SPLINE
SPL {X  -123.821, Y  +785.537, Z    +0.000, E1   -64.536, E3 +26761.912}
SPL {X  -153.467, Y  +737.853, Z    +0.000, E1   -51.757, E3 +26764.227}
SPL {X  -161.000, Y  +714.475, Z    +0.000, E1   -39.424, E3 +26763.699}
SPL {X  -164.534, Y  +694.695, Z    +0.000, E1   -23.511, E3 +26761.989}
SPL {X  -165.597, Y  +679.703, Z    +0.000, E1    -7.645, E3 +26761.865}
SPL {X  -165.650, Y  +673.520, Z    +0.000, E1    -0.048, E3 +26760.817}
SPL {X  -165.650, Y  +671.692, Z    +0.000, E1    +4.450, E3 +26760.383}
SPL {X  -165.650, Y  +667.743, Z    +0.000, E1   +15.617, E3 +26760.301}
SPL {X  -165.650, Y  +662.891, Z    +0.000, E1   +29.740, E3 +26759.819}
SPL {X  -165.650, Y  +658.373, Z    +0.000, E1   +40.877, E3 +26760.016}
SPL {X  -165.650, Y  +650.834, Z    +0.000, E1   +55.143, E3 +26759.270}
SPL {X  -165.650, Y  +639.785, Z    +0.000, E1   +67.512, E3 +26758.487}
SPL {X  -165.650, Y  +619.979, Z    +0.000, E1   +79.465, E3 +26754.656}
SPL {X  -165.650, Y  +584.722, Z    +0.000, E1   +79.551, E3 +26763.947}
SPL {X  -165.650, Y  +560.326, Z    +0.000, E1   +78.360, E3 +26773.669}
SPL {X  -160.258, Y  +336.579, Z    +0.000, E1   +78.314, E3 +26845.191}
SPL {X  -159.618, Y  +334.207, Z    +0.000, E1   +75.622, E3 +26876.005}
SPL {X  -156.487, Y  +324.170, Z    +0.000, E1   +75.150, E3 +26886.360}
SPL {X  -142.256, Y  +293.629, Z    +0.000, E1   +77.020, E3 +26881.460}
ENDSPLINE

SPLINE
SPL {X  -142.811, Y  +294.566, Z    +0.000, E1   +75.668, E3 +26893.422}
ENDSPLINE

SPLINE
SPL {X  -141.646, Y  +292.615, Z    +0.000, E1   +74.702, E3 +26902.516}
SPL {X  -140.419, Y  +290.622, Z    +0.000, E1   +73.705, E3 +26911.359}
SPL {X  -136.008, Y  +283.940, Z    +0.000, E1   +73.594, E3 +26915.478}
SPL {X  -132.748, Y  +279.415, Z    +0.000, E1   +73.006, E3 +26921.534}
SPL {X  -129.007, Y  +274.590, Z    +0.000, E1   +72.484, E3 +26926.883}
SPL {X  -125.914, Y  +270.864, Z    +0.000, E1   +72.144, E3 +26930.375}
SPL {X  -123.729, Y  +268.359, Z    +0.000, E1   +71.932, E3 +26932.547}
SPL {X  -111.023, Y  +255.562, Z    +0.000, E1   +75.772, E3 +26923.413}
SPL {X   -49.289, Y  +220.353, Z    +0.000, E1   +56.690, E3 +27116.128}
ENDSPLINE

SPLINE
SPL {X  -127.117, Y  +272.287, Z    +0.000, E1   +62.713, E3 +27285.350}
SPL {X  -154.956, Y  +319.945, Z    +0.000, E1   +49.402, E3 +27289.749}
SPL {X  -162.871, Y  +348.286, Z    +0.000, E1   +32.462, E3 +27288.776}
SPL {X  -165.127, Y  +365.342, Z    +0.000, E1   +17.250, E3 +27288.615}
SPL {X  -165.640, Y  +376.693, Z    +0.000, E1    +4.721, E3 +27288.188}
SPL {X  -165.650, Y  +380.500, Z    +0.000, E1    -0.000, E3 +27287.339}
SPL {X  -165.650, Y  +382.123, Z    +0.000, E1    -3.912, E3 +27286.966}
SPL {X  -165.650, Y  +387.069, Z    +0.000, E1   -17.420, E3 +27286.677}
SPL {X  -165.650, Y  +393.439, Z    +0.000, E1   -35.398, E3 +27286.223}
SPL {X  -165.650, Y  +400.610, Z    +0.000, E1   -50.510, E3 +27285.961}
SPL {X  -165.650, Y  +414.376, Z    +0.000, E1   -68.098, E3 +27283.994}
SPL {X  -165.650, Y  +468.582, Z    +0.000, E1   -78.237, E3 +27292.765}
SPL {X  -160.244, Y  +717.475, Z    +0.000, E1   -78.917, E3 +27365.322}
SPL {X  -159.651, Y  +719.676, Z    +0.000, E1   -75.661, E3 +27401.709}
SPL {X  -157.156, Y  +727.862, Z    +0.000, E1   -75.175, E3 +27411.191}
SPL {X  -154.068, Y  +736.353, Z    +0.000, E1   -74.906, E3 +27418.366}
SPL {X  -149.738, Y  +746.340, Z    +0.000, E1   -74.451, E3 +27428.054}
SPL {X  -144.163, Y  +757.090, Z    +0.000, E1   -74.033, E3 +27437.146}
SPL {X  -139.284, Y  +765.165, Z    +0.000, E1   -73.322, E3 +27446.841}
SPL {X  -134.662, Y  +771.969, Z    +0.000, E1   -72.884, E3 +27453.173}
SPL {X  -131.459, Y  +776.289, Z    +0.000, E1   -72.475, E3 +27457.840}
SPL {X  -127.605, Y  +781.126, Z    +0.000, E1   -71.922, E3 +27463.284}
SPL {X  -124.773, Y  +784.457, Z    +0.000, E1   -71.383, E3 +27467.331}
SPL {X  -119.086, Y  +790.645, Z    +0.000, E1   -72.931, E3 +27464.185}
SPL {X   -51.449, Y  +832.958, Z    +0.000, E1   -57.230, E3 +27621.705}
ENDSPLINE

SPLINE
SPL {X  -123.821, Y  +785.537, Z    +0.000, E1   -64.536, E3 +27823.450}
SPL {X  -153.467, Y  +737.853, Z    +0.000, E1   -51.757, E3 +27825.765}
SPL {X  -161.000, Y  +714.475, Z    +0.000, E1   -39.424, E3 +27825.238}
SPL {X  -164.534, Y  +694.695, Z    +0.000, E1   -23.511, E3 +27823.528}
SPL {X  -165.597, Y  +679.703, Z    +0.000, E1    -7.645, E3 +27823.403}
SPL {X  -165.650, Y  +673.520, Z    +0.000, E1    -0.048, E3 +27822.355}
SPL {X  -165.650, Y  +671.692, Z    +0.000, E1    +4.450, E3 +27821.922}
SPL {X  -165.650, Y  +667.743, Z    +0.000, E1   +15.617, E3 +27821.840}
SPL {X  -165.650, Y  +661.459, Z    +0.000, E1   +33.218, E3 +27821.420}
SPL {X  -165.650, Y  +653.296, Z    +0.000, E1   +51.333, E3 +27820.975}
SPL {X  -165.650, Y  +642.000, Z    +0.000, E1   +65.561, E3 +27820.188}
SPL {X  -165.650, Y  +619.979, Z    +0.000, E1   +79.465, E3 +27816.194}
SPL {X  -165.650, Y  +569.632, Z    +0.000, E1   +78.783, E3 +27831.473}
SPL {X  -158.840, Y  +331.491, Z    +0.000, E1   +77.462, E3 +27917.783}
ENDSPLINE

SPLINE
SPL {X  -159.893, Y  +335.208, Z    +0.000, E1   +75.483, E3 +27938.518}
ENDSPLINE

SPLINE
SPL {X  -156.487, Y  +324.170, Z    +0.000, E1   +75.150, E3 +27947.899}
SPL {X  -142.256, Y  +293.629, Z    +0.000, E1   +77.020, E3 +27942.999}
ENDSPLINE

SPLINE
SPL {X  -142.811, Y  +294.566, Z    +0.000, E1   +75.668, E3 +27954.961}
ENDSPLINE

SPLINE
SPL {X  -141.646, Y  +292.615, Z    +0.000, E1   +74.702, E3 +27964.055}
SPL {X  -140.419, Y  +290.622, Z    +0.000, E1   +73.705, E3 +27972.898}
SPL {X  -136.008, Y  +283.940, Z    +0.000, E1   +73.594, E3 +27977.017}
SPL {X  -132.748, Y  +279.415, Z    +0.000, E1   +73.006, E3 +27983.073}
SPL {X  -129.007, Y  +274.590, Z    +0.000, E1   +72.484, E3 +27988.421}
SPL {X  -125.914, Y  +270.864, Z    +0.000, E1   +72.144, E3 +27991.913}
SPL {X  -123.729, Y  +268.359, Z    +0.000, E1   +71.932, E3 +27994.085}
SPL {X  -111.023, Y  +255.562, Z    +0.000, E1   +75.772, E3 +27984.951}
SPL {X   -49.289, Y  +220.353, Z    +0.000, E1   +56.690, E3 +28177.666}
ENDSPLINE

SPLINE
SPL {X  -127.117, Y  +272.287, Z    +0.000, E1   +62.713, E3 +28346.888}
SPL {X  -154.956, Y  +319.945, Z    +0.000, E1   +49.402, E3 +28351.287}
SPL {X  -162.871, Y  +348.286, Z    +0.000, E1   +32.462, E3 +28350.315}
SPL {X  -165.127, Y  +365.342, Z    +0.000, E1   +17.250, E3 +28350.153}
SPL {X  -165.640, Y  +376.693, Z    +0.000, E1    +4.721, E3 +28349.726}
SPL {X  -165.650, Y  +380.500, Z    +0.000, E1    -0.000, E3 +28348.877}
SPL {X  -165.650, Y  +383.262, Z    +0.000, E1    -6.645, E3 +28348.406}
SPL {X  -165.650, Y  +388.390, Z    +0.000, E1   -21.508, E3 +28348.194}
SPL {X  -165.650, Y  +393.439, Z    +0.000, E1   -35.398, E3 +28347.762}
SPL {X  -165.650, Y  +400.610, Z    +0.000, E1   -50.510, E3 +28347.499}
SPL {X  -165.650, Y  +414.376, Z    +0.000, E1   -68.098, E3 +28345.533}
SPL {X  -165.650, Y  +468.582, Z    +0.000, E1   -78.237, E3 +28354.303}
SPL {X  -158.306, Y  +724.277, Z    +0.000, E1   -77.461, E3 +28444.744}
ENDSPLINE

SPLINE
SPL {X  -160.145, Y  +717.851, Z    +0.000, E1   -75.386, E3 +28465.258}
ENDSPLINE

SPLINE
SPL {X  -157.156, Y  +727.862, Z    +0.000, E1   -75.175, E3 +28472.730}
SPL {X  -154.068, Y  +736.353, Z    +0.000, E1   -74.906, E3 +28479.905}
SPL {X  -149.738, Y  +746.340, Z    +0.000, E1   -74.451, E3 +28489.592}
SPL {X  -144.163, Y  +757.090, Z    +0.000, E1   -74.033, E3 +28498.685}
SPL {X  -140.473, Y  +763.291, Z    +0.000, E1   -73.478, E3 +28506.126}
SPL {X  -135.914, Y  +770.196, Z    +0.000, E1   -72.974, E3 +28513.302}
SPL {X  -131.459, Y  +776.289, Z    +0.000, E1   -72.475, E3 +28519.378}
SPL {X  -128.771, Y  +779.702, Z    +0.000, E1   -71.875, E3 +28524.325}
SPL {X  -124.506, Y  +784.762, Z    +0.000, E1   -71.815, E3 +28527.213}
SPL {X  -112.958, Y  +796.663, Z    +0.000, E1   -74.119, E3 +28523.917}
SPL {X   -51.449, Y  +832.958, Z    +0.000, E1   -57.230, E3 +28683.244}
ENDSPLINE

SPLINE
SPL {X  -123.821, Y  +785.537, Z    +0.000, E1   -64.536, E3 +28884.989}
SPL {X  -153.467, Y  +737.853, Z    +0.000, E1   -51.757, E3 +28887.304}
SPL {X  -162.176, Y  +709.248, Z    +0.000, E1   -35.773, E3 +28886.329}
SPL {X  -164.888, Y  +691.368, Z    +0.000, E1   -20.174, E3 +28884.767}
SPL {X  -165.597, Y  +679.703, Z    +0.000, E1    -7.645, E3 +28884.942}
SPL {X  -165.650, Y  +673.520, Z    +0.000, E1    -0.048, E3 +28883.894}
SPL {X  -165.650, Y  +671.692, Z    +0.000, E1    +4.450, E3 +28883.460}
SPL {X  -165.650, Y  +667.743, Z    +0.000, E1   +15.617, E3 +28883.378}
SPL {X  -165.650, Y  +661.459, Z    +0.000, E1   +33.218, E3 +28882.959}
SPL {X  -165.650, Y  +650.834, Z    +0.000, E1   +55.143, E3 +28882.347}
SPL {X  -165.650, Y  +639.785, Z    +0.000, E1   +67.512, E3 +28881.564}
SPL {X  -165.650, Y  +619.979, Z    +0.000, E1   +79.465, E3 +28877.733}
SPL {X  -165.650, Y  +569.632, Z    +0.000, E1   +78.783, E3 +28893.011}
SPL {X  -158.840, Y  +331.491, Z    +0.000, E1   +77.462, E3 +28979.322}
ENDSPLINE

SPLINE
SPL {X  -159.893, Y  +335.208, Z    +0.000, E1   +75.483, E3 +29000.056}
ENDSPLINE

SPLINE
SPL {X  -156.487, Y  +324.170, Z    +0.000, E1   +75.150, E3 +29009.437}
SPL {X  -142.256, Y  +293.629, Z    +0.000, E1   +77.020, E3 +29004.537}
ENDSPLINE

SPLINE
SPL {X  -142.811, Y  +294.566, Z    +0.000, E1   +75.668, E3 +29016.499}
ENDSPLINE

SPLINE
SPL {X  -141.646, Y  +292.615, Z    +0.000, E1   +74.702, E3 +29025.593}
SPL {X  -140.419, Y  +290.622, Z    +0.000, E1   +73.705, E3 +29034.436}
SPL {X  -136.008, Y  +283.940, Z    +0.000, E1   +73.594, E3 +29038.555}
SPL {X  -132.748, Y  +279.415, Z    +0.000, E1   +73.006, E3 +29044.611}
SPL {X  -129.007, Y  +274.590, Z    +0.000, E1   +72.484, E3 +29049.960}
SPL {X  -125.914, Y  +270.864, Z    +0.000, E1   +72.144, E3 +29053.451}
SPL {X  -123.729, Y  +268.359, Z    +0.000, E1   +71.932, E3 +29055.624}
SPL {X  -111.023, Y  +255.562, Z    +0.000, E1   +75.772, E3 +29046.490}
SPL {X   -49.289, Y  +220.353, Z    +0.000, E1   +56.690, E3 +29239.205}
ENDSPLINE

SPLINE
SPL {X  -127.117, Y  +272.287, Z    +0.000, E1   +62.713, E3 +29408.427}
SPL {X  -152.442, Y  +313.682, Z    +0.000, E1   +51.943, E3 +29412.658}
SPL {X  -162.319, Y  +345.447, Z    +0.000, E1   +34.671, E3 +29412.084}
SPL {X  -165.127, Y  +365.342, Z    +0.000, E1   +17.250, E3 +29411.692}
SPL {X  -165.640, Y  +376.693, Z    +0.000, E1    +4.721, E3 +29411.265}
SPL {X  -165.650, Y  +380.500, Z    +0.000, E1    -0.000, E3 +29410.416}
SPL {X  -165.650, Y  +383.262, Z    +0.000, E1    -6.645, E3 +29409.945}
SPL {X  -165.650, Y  +388.390, Z    +0.000, E1   -21.508, E3 +29409.733}
SPL {X  -165.650, Y  +393.439, Z    +0.000, E1   -35.398, E3 +29409.300}
SPL {X  -165.650, Y  +400.610, Z    +0.000, E1   -50.510, E3 +29409.038}
SPL {X  -165.650, Y  +414.376, Z    +0.000, E1   -68.098, E3 +29407.071}
SPL {X  -165.650, Y  +459.729, Z    +0.000, E1   -78.035, E3 +29413.526}
SPL {X  -165.650, Y  +475.450, Z    +0.000, E1   -78.345, E3 +29417.640}
SPL {X  -158.306, Y  +724.277, Z    +0.000, E1   -77.461, E3 +29506.283}
ENDSPLINE

SPLINE
SPL {X  -160.145, Y  +717.851, Z    +0.000, E1   -75.386, E3 +29526.796}
ENDSPLINE

SPLINE
SPL {X  -157.156, Y  +727.862, Z    +0.000, E1   -75.175, E3 +29534.268}
SPL {X  -154.068, Y  +736.353, Z    +0.000, E1   -74.906, E3 +29541.443}
SPL {X  -149.738, Y  +746.340, Z    +0.000, E1   -74.451, E3 +29551.131}
SPL {X  -145.204, Y  +755.223, Z    +0.000, E1   -74.188, E3 +29557.857}
SPL {X  -141.453, Y  +761.704, Z    +0.000, E1   -73.638, E3 +29565.779}
SPL {X  -135.914, Y  +770.196, Z    +0.000, E1   -72.974, E3 +29574.841}
SPL {X  -131.459, Y  +776.289, Z    +0.000, E1   -72.475, E3 +29580.917}
SPL {X  -128.771, Y  +779.702, Z    +0.000, E1   -71.875, E3 +29585.863}
SPL {X  -124.506, Y  +784.762, Z    +0.000, E1   -71.815, E3 +29588.752}
SPL {X  -112.958, Y  +796.663, Z    +0.000, E1   -74.119, E3 +29585.455}
SPL {X   -51.449, Y  +832.958, Z    +0.000, E1   -57.230, E3 +29744.782}
ENDSPLINE

SPLINE
SPL {X  -123.821, Y  +785.537, Z    +0.000, E1   -64.536, E3 +29946.527}
SPL {X  -153.467, Y  +737.853, Z    +0.000, E1   -51.757, E3 +29948.842}
SPL {X  -162.176, Y  +709.248, Z    +0.000, E1   -35.773, E3 +29947.868}
SPL {X  -164.888, Y  +691.368, Z    +0.000, E1   -20.174, E3 +29946.305}
SPL {X  -165.597, Y  +679.703, Z    +0.000, E1    -7.645, E3 +29946.480}
SPL {X  -165.650, Y  +673.520, Z    +0.000, E1    -0.048, E3 +29945.432}
SPL {X  -165.650, Y  +671.692, Z    +0.000, E1    +4.450, E3 +29944.999}
SPL {X  -165.650, Y  +667.743, Z    +0.000, E1   +15.617, E3 +29944.917}
SPL {X  -165.650, Y  +661.459, Z    +0.000, E1   +33.218, E3 +29944.497}
SPL {X  -165.650, Y  +653.296, Z    +0.000, E1   +51.333, E3 +29944.052}
SPL {X  -165.650, Y  +642.000, Z    +0.000, E1   +65.561, E3 +29943.265}
SPL {X  -165.650, Y  +619.979, Z    +0.000, E1   +79.465, E3 +29939.271}
SPL {X  -165.650, Y  +569.632, Z    +0.000, E1   +78.783, E3 +29954.550}
SPL {X  -158.840, Y  +331.491, Z    +0.000, E1   +77.462, E3 +30040.860}
ENDSPLINE

SPLINE
SPL {X  -159.893, Y  +335.208, Z    +0.000, E1   +75.483, E3 +30061.595}
ENDSPLINE

SPLINE
SPL {X  -156.487, Y  +324.170, Z    +0.000, E1   +75.150, E3 +30070.976}
SPL {X  -142.256, Y  +293.629, Z    +0.000, E1   +77.020, E3 +30066.076}
ENDSPLINE

SPLINE
SPL {X  -142.811, Y  +294.566, Z    +0.000, E1   +75.668, E3 +30078.038}
ENDSPLINE

SPLINE
SPL {X  -141.646, Y  +292.615, Z    +0.000, E1   +74.702, E3 +30087.131}
SPL {X  -140.419, Y  +290.622, Z    +0.000, E1   +73.705, E3 +30095.975}
SPL {X  -135.839, Y  +283.697, Z    +0.000, E1   +73.388, E3 +30101.713}
SPL {X  -131.336, Y  +277.551, Z    +0.000, E1   +72.879, E3 +30107.965}
SPL {X  -126.848, Y  +271.966, Z    +0.000, E1   +72.322, E3 +30113.693}
SPL {X  -123.729, Y  +268.359, Z    +0.000, E1   +71.932, E3 +30117.162}
SPL {X  -111.023, Y  +255.562, Z    +0.000, E1   +75.772, E3 +30108.028}
SPL {X   -52.752, Y  +221.474, Z    +0.000, E1   +59.157, E3 +30237.280}
SPL {X   -49.901, Y  +220.545, Z    +0.000, E1   +56.696, E3 +30323.672}
ENDSPLINE

SPLINE
SPL {X  -127.117, Y  +272.287, Z    +0.000, E1   +62.713, E3 +30469.965}
SPL {X  -152.442, Y  +313.682, Z    +0.000, E1   +51.943, E3 +30474.197}
SPL {X  -162.319, Y  +345.447, Z    +0.000, E1   +34.671, E3 +30473.622}
SPL {X  -165.127, Y  +365.342, Z    +0.000, E1   +17.250, E3 +30473.230}
SPL {X  -165.640, Y  +376.693, Z    +0.000, E1    +4.721, E3 +30472.803}
SPL {X  -165.650, Y  +380.500, Z    +0.000, E1    -0.000, E3 +30471.954}
SPL {X  -165.650, Y  +382.123, Z    +0.000, E1    -3.912, E3 +30471.581}
SPL {X  -165.650, Y  +387.069, Z    +0.000, E1   -17.420, E3 +30471.293}
SPL {X  -165.650, Y  +393.439, Z    +0.000, E1   -35.398, E3 +30470.839}
SPL {X  -165.650, Y  +400.610, Z    +0.000, E1   -50.510, E3 +30470.576}
SPL {X  -165.650, Y  +414.376, Z    +0.000, E1   -68.098, E3 +30468.610}
SPL {X  -165.650, Y  +468.582, Z    +0.000, E1   -78.237, E3 +30477.380}
SPL {X  -160.244, Y  +717.475, Z    +0.000, E1   -78.917, E3 +30549.938}
SPL {X  -159.651, Y  +719.676, Z    +0.000, E1   -75.661, E3 +30586.324}
SPL {X  -157.156, Y  +727.862, Z    +0.000, E1   -75.175, E3 +30595.807}
SPL {X  -154.068, Y  +736.353, Z    +0.000, E1   -74.906, E3 +30602.981}
SPL {X  -149.738, Y  +746.340, Z    +0.000, E1   -74.451, E3 +30612.669}
SPL {X  -144.163, Y  +757.090, Z    +0.000, E1   -74.033, E3 +30621.762}
SPL {X  -139.284, Y  +765.165, Z    +0.000, E1   -73.322, E3 +30631.456}
SPL {X  -134.662, Y  +771.969, Z    +0.000, E1   -72.884, E3 +30637.788}
SPL {X  -131.459, Y  +776.289, Z    +0.000, E1   -72.475, E3 +30642.455}
SPL {X  -127.605, Y  +781.126, Z    +0.000, E1   -71.922, E3 +30647.899}
SPL {X  -124.773, Y  +784.457, Z    +0.000, E1   -71.383, E3 +30651.947}
SPL {X  -119.086, Y  +790.645, Z    +0.000, E1   -72.931, E3 +30648.801}
SPL {X   -51.449, Y  +832.958, Z    +0.000, E1   -57.230, E3 +30806.321}
ENDSPLINE

SPLINE
SPL {X  -123.821, Y  +785.537, Z    +0.000, E1   -64.536, E3 +31008.066}
SPL {X  -153.467, Y  +737.853, Z    +0.000, E1   -51.757, E3 +31010.381}
SPL {X  -161.000, Y  +714.475, Z    +0.000, E1   -39.424, E3 +31009.853}
SPL {X  -164.534, Y  +694.695, Z    +0.000, E1   -23.511, E3 +31008.143}
SPL {X  -165.597, Y  +679.703, Z    +0.000, E1    -7.645, E3 +31008.019}
SPL {X  -165.650, Y  +673.520, Z    +0.000, E1    -0.048, E3 +31006.971}
SPL {X  -165.650, Y  +671.692, Z    +0.000, E1    +4.450, E3 +31006.537}
SPL {X  -165.650, Y  +667.743, Z    +0.000, E1   +15.617, E3 +31006.455}
SPL {X  -165.650, Y  +661.459, Z    +0.000, E1   +33.218, E3 +31006.035}
SPL {X  -165.650, Y  +653.296, Z    +0.000, E1   +51.333, E3 +31005.591}
SPL {X  -165.650, Y  +642.000, Z    +0.000, E1   +65.561, E3 +31004.803}
SPL {X  -165.650, Y  +619.979, Z    +0.000, E1   +79.465, E3 +31000.810}
SPL {X  -165.650, Y  +569.632, Z    +0.000, E1   +78.783, E3 +31016.088}
SPL {X  -158.840, Y  +331.491, Z    +0.000, E1   +77.462, E3 +31102.398}
ENDSPLINE

SPLINE
SPL {X  -159.893, Y  +335.208, Z    +0.000, E1   +75.483, E3 +31123.133}
ENDSPLINE

SPLINE
SPL {X  -156.487, Y  +324.170, Z    +0.000, E1   +75.150, E3 +31132.514}
SPL {X  -142.256, Y  +293.629, Z    +0.000, E1   +77.020, E3 +31127.614}
ENDSPLINE

SPLINE
SPL {X  -142.811, Y  +294.566, Z    +0.000, E1   +75.668, E3 +31139.576}
ENDSPLINE

SPLINE
SPL {X  -141.646, Y  +292.615, Z    +0.000, E1   +74.702, E3 +31148.670}
SPL {X  -140.419, Y  +290.622, Z    +0.000, E1   +73.705, E3 +31157.513}
SPL {X  -136.008, Y  +283.940, Z    +0.000, E1   +73.594, E3 +31161.632}
SPL {X  -132.748, Y  +279.415, Z    +0.000, E1   +73.006, E3 +31167.688}
SPL {X  -129.007, Y  +274.590, Z    +0.000, E1   +72.484, E3 +31173.037}
SPL {X  -125.914, Y  +270.864, Z    +0.000, E1   +72.144, E3 +31176.528}
SPL {X  -123.729, Y  +268.359, Z    +0.000, E1   +71.932, E3 +31178.701}
SPL {X  -111.023, Y  +255.562, Z    +0.000, E1   +75.772, E3 +31169.567}
SPL {X   -49.289, Y  +220.353, Z    +0.000, E1   +56.690, E3 +31362.282}
ENDSPLINE

SPLINE
SPL {X  -127.117, Y  +272.287, Z    +0.000, E1   +62.713, E3 +31531.503}
SPL {X  -154.956, Y  +319.945, Z    +0.000, E1   +49.402, E3 +31535.903}
SPL {X  -162.871, Y  +348.286, Z    +0.000, E1   +32.462, E3 +31534.930}
SPL {X  -165.127, Y  +365.342, Z    +0.000, E1   +17.250, E3 +31534.769}
SPL {X  -165.640, Y  +376.693, Z    +0.000, E1    +4.721, E3 +31534.342}
SPL {X  -165.650, Y  +380.500, Z    +0.000, E1    -0.000, E3 +31533.493}
SPL {X  -165.650, Y  +382.123, Z    +0.000, E1    -3.912, E3 +31533.120}
SPL {X  -165.650, Y  +387.069, Z    +0.000, E1   -17.420, E3 +31532.831}
SPL {X  -165.650, Y  +393.439, Z    +0.000, E1   -35.398, E3 +31532.377}
SPL {X  -165.650, Y  +402.896, Z    +0.000, E1   -54.480, E3 +31531.618}
SPL {X  -165.650, Y  +416.934, Z    +0.000, E1   -69.887, E3 +31530.084}
SPL {X  -165.650, Y  +459.729, Z    +0.000, E1   -78.035, E3 +31536.603}
SPL {X  -165.650, Y  +475.450, Z    +0.000, E1   -78.345, E3 +31540.717}
SPL {X  -160.244, Y  +717.475, Z    +0.000, E1   -78.917, E3 +31611.476}
SPL {X  -159.651, Y  +719.676, Z    +0.000, E1   -75.661, E3 +31647.863}
SPL {X  -157.156, Y  +727.862, Z    +0.000, E1   -75.175, E3 +31657.345}
SPL {X  -154.068, Y  +736.353, Z    +0.000, E1   -74.906, E3 +31664.520}
SPL {X  -149.738, Y  +746.340, Z    +0.000, E1   -74.451, E3 +31674.208}
SPL {X  -144.163, Y  +757.090, Z    +0.000, E1   -74.033, E3 +31683.300}
SPL {X  -139.284, Y  +765.165, Z    +0.000, E1   -73.322, E3 +31692.995}
SPL {X  -134.662, Y  +771.969, Z    +0.000, E1   -72.884, E3 +31699.326}
SPL {X  -131.459, Y  +776.289, Z    +0.000, E1   -72.475, E3 +31703.994}
SPL {X  -128.771, Y  +779.702, Z    +0.000, E1   -71.875, E3 +31708.940}
SPL {X  -125.267, Y  +783.889, Z    +0.000, E1   -71.674, E3 +31712.053}
SPL {X  -119.086, Y  +790.645, Z    +0.000, E1   -72.931, E3 +31710.339}
SPL {X   -51.449, Y  +832.958, Z    +0.000, E1   -57.230, E3 +31867.859}
ENDSPLINE

SPLINE
SPL {X  -123.821, Y  +785.537, Z    +0.000, E1   -64.536, E3 +32069.604}
SPL {X  -153.467, Y  +737.853, Z    +0.000, E1   -51.757, E3 +32071.919}
SPL {X  -162.176, Y  +709.248, Z    +0.000, E1   -35.773, E3 +32070.945}
SPL {X  -164.888, Y  +691.368, Z    +0.000, E1   -20.174, E3 +32069.382}
SPL {X  -165.597, Y  +679.703, Z    +0.000, E1    -7.645, E3 +32069.557}
SPL {X  -165.650, Y  +673.520, Z    +0.000, E1    -0.048, E3 +32068.509}
SPL {X  -165.650, Y  +671.692, Z    +0.000, E1    +4.450, E3 +32068.076}
SPL {X  -165.650, Y  +667.743, Z    +0.000, E1   +15.617, E3 +32067.994}
SPL {X  -165.650, Y  +661.459, Z    +0.000, E1   +33.218, E3 +32067.574}
SPL {X  -165.650, Y  +653.296, Z    +0.000, E1   +51.333, E3 +32067.129}
SPL {X  -165.650, Y  +642.000, Z    +0.000, E1   +65.561, E3 +32066.341}
SPL {X  -165.650, Y  +619.979, Z    +0.000, E1   +79.465, E3 +32062.348}
SPL {X  -165.650, Y  +584.722, Z    +0.000, E1   +79.551, E3 +32071.639}
SPL {X  -165.650, Y  +560.326, Z    +0.000, E1   +78.360, E3 +32081.361}
SPL {X  -158.840, Y  +331.491, Z    +0.000, E1   +77.462, E3 +32163.937}
ENDSPLINE

SPLINE
SPL {X  -159.893, Y  +335.208, Z    +0.000, E1   +75.483, E3 +32184.672}
ENDSPLINE

SPLINE
SPL {X  -156.487, Y  +324.170, Z    +0.000, E1   +75.150, E3 +32194.053}
SPL {X  -142.256, Y  +293.629, Z    +0.000, E1   +77.020, E3 +32189.152}
ENDSPLINE

SPLINE
SPL {X  -142.811, Y  +294.566, Z    +0.000, E1   +75.668, E3 +32201.115}
ENDSPLINE

SPLINE
SPL {X  -141.646, Y  +292.615, Z    +0.000, E1   +74.702, E3 +32210.208}
SPL {X  -140.419, Y  +290.622, Z    +0.000, E1   +73.705, E3 +32219.052}
SPL {X  -136.008, Y  +283.940, Z    +0.000, E1   +73.594, E3 +32223.171}
SPL {X  -132.748, Y  +279.415, Z    +0.000, E1   +73.006, E3 +32229.226}
SPL {X  -129.007, Y  +274.590, Z    +0.000, E1   +72.484, E3 +32234.575}
SPL {X  -125.914, Y  +270.864, Z    +0.000, E1   +72.144, E3 +32238.067}
SPL {X  -123.729, Y  +268.359, Z    +0.000, E1   +71.932, E3 +32240.239}
SPL {X  -111.023, Y  +255.562, Z    +0.000, E1   +75.772, E3 +32231.105}
SPL {X   -49.289, Y  +220.353, Z    +0.000, E1   +56.690, E3 +32423.820}
ENDSPLINE

SPLINE
SPL {X  -127.117, Y  +272.287, Z    +0.000, E1   +62.713, E3 +32593.042}
SPL {X  -152.442, Y  +313.682, Z    +0.000, E1   +51.943, E3 +32597.274}
SPL {X  -159.925, Y  +335.326, Z    +0.000, E1   +41.361, E3 +32597.216}
SPL {X  -163.450, Y  +351.595, Z    +0.000, E1   +29.785, E3 +32596.327}
SPL {X  -165.127, Y  +365.342, Z    +0.000, E1   +17.250, E3 +32596.307}
SPL {X  -165.640, Y  +376.693, Z    +0.000, E1    +4.721, E3 +32595.880}
SPL {X  -165.650, Y  +380.500, Z    +0.000, E1    -0.000, E3 +32595.031}
SPL {X  -165.650, Y  +382.123, Z    +0.000, E1    -3.912, E3 +32594.658}
SPL {X  -165.650, Y  +387.069, Z    +0.000, E1   -17.420, E3 +32594.370}
SPL {X  -165.650, Y  +393.439, Z    +0.000, E1   -35.398, E3 +32593.915}
SPL {X  -165.650, Y  +400.610, Z    +0.000, E1   -50.510, E3 +32593.653}
SPL {X  -165.650, Y  +414.376, Z    +0.000, E1   -68.098, E3 +32591.687}
SPL {X  -165.650, Y  +468.582, Z    +0.000, E1   -78.237, E3 +32600.457}
SPL {X  -160.244, Y  +717.475, Z    +0.000, E1   -78.917, E3 +32673.015}
SPL {X  -159.651, Y  +719.676, Z    +0.000, E1   -75.661, E3 +32709.401}
SPL {X  -157.156, Y  +727.862, Z    +0.000, E1   -75.175, E3 +32718.884}
SPL {X  -152.814, Y  +739.436, Z    +0.000, E1   -74.813, E3 +32728.737}
SPL {X  -148.754, Y  +748.385, Z    +0.000, E1   -74.281, E3 +32738.180}
SPL {X  -144.163, Y  +757.090, Z    +0.000, E1   -74.033, E3 +32744.838}
SPL {X  -140.473, Y  +763.291, Z    +0.000, E1   -73.478, E3 +32752.280}
SPL {X  -135.914, Y  +770.196, Z    +0.000, E1   -72.974, E3 +32759.456}
SPL {X  -131.459, Y  +776.289, Z    +0.000, E1   -72.475, E3 +32765.532}
SPL {X  -128.771, Y  +779.702, Z    +0.000, E1   -71.875, E3 +32770.479}
SPL {X  -125.267, Y  +783.889, Z    +0.000, E1   -71.674, E3 +32773.591}
SPL {X  -119.086, Y  +790.645, Z    +0.000, E1   -72.931, E3 +32771.878}
SPL {X   -51.449, Y  +832.958, Z    +0.000, E1   -57.230, E3 +32929.398}
ENDSPLINE

SPLINE
SPL {X  -123.821, Y  +785.537, Z    +0.000, E1   -64.536, E3 +33131.143}
SPL {X  -153.467, Y  +737.853, Z    +0.000, E1   -51.757, E3 +33133.458}
SPL {X  -161.000, Y  +714.475, Z    +0.000, E1   -39.424, E3 +33132.930}
SPL {X  -164.534, Y  +694.695, Z    +0.000, E1   -23.511, E3 +33131.220}
SPL {X  -165.597, Y  +679.703, Z    +0.000, E1    -7.645, E3 +33131.096}
SPL {X  -165.650, Y  +673.520, Z    +0.000, E1    -0.048, E3 +33130.048}
SPL {X  -165.650, Y  +671.692, Z    +0.000, E1    +4.450, E3 +33129.614}
SPL {X  -165.650, Y  +667.743, Z    +0.000, E1   +15.617, E3 +33129.532}
SPL {X  -165.650, Y  +662.891, Z    +0.000, E1   +29.740, E3 +33129.050}
SPL {X  -165.650, Y  +655.319, Z    +0.000, E1   +47.265, E3 +33128.899}
SPL {X  -165.650, Y  +642.000, Z    +0.000, E1   +65.561, E3 +33127.880}
SPL {X  -165.650, Y  +619.979, Z    +0.000, E1   +79.465, E3 +33123.886}
SPL {X  -165.650, Y  +569.632, Z    +0.000, E1   +78.783, E3 +33139.165}
SPL {X  -158.840, Y  +331.491, Z    +0.000, E1   +77.462, E3 +33225.475}
ENDSPLINE

SPLINE
SPL {X  -159.893, Y  +335.208, Z    +0.000, E1   +75.483, E3 +33246.210}
ENDSPLINE

SPLINE
SPL {X  -156.487, Y  +324.170, Z    +0.000, E1   +75.150, E3 +33255.591}
SPL {X  -142.256, Y  +293.629, Z    +0.000, E1   +77.020, E3 +33250.691}
ENDSPLINE

SPLINE
SPL {X  -142.811, Y  +294.566, Z    +0.000, E1   +75.668, E3 +33262.653}
ENDSPLINE

SPLINE
SPL {X  -141.646, Y  +292.615, Z    +0.000, E1   +74.702, E3 +33271.747}
SPL {X  -140.419, Y  +290.622, Z    +0.000, E1   +73.705, E3 +33280.590}
SPL {X  -135.839, Y  +283.697, Z    +0.000, E1   +73.388, E3 +33286.328}
SPL {X  -131.903, Y  +278.292, Z    +0.000, E1   +73.096, E3 +33290.818}
SPL {X  -129.007, Y  +274.590, Z    +0.000, E1   +72.484, E3 +33296.114}
SPL {X  -124.646, Y  +269.397, Z    +0.000, E1   +72.041, E3 +33300.862}
SPL {X  -111.023, Y  +255.562, Z    +0.000, E1   +75.772, E3 +33292.644}
SPL {X   -49.289, Y  +220.353, Z    +0.000, E1   +56.690, E3 +33485.358}
ENDSPLINE

SPLINE
SPL {X  -127.117, Y  +272.287, Z    +0.000, E1   +62.713, E3 +33654.580}
SPL {X  -154.956, Y  +319.945, Z    +0.000, E1   +49.402, E3 +33658.979}
SPL {X  -162.871, Y  +348.286, Z    +0.000, E1   +32.462, E3 +33658.007}
SPL {X  -165.127, Y  +365.342, Z    +0.000, E1   +17.250, E3 +33657.846}
SPL {X  -165.640, Y  +376.693, Z    +0.000, E1    +4.721, E3 +33657.419}
SPL {X  -165.650, Y  +380.500, Z    +0.000, E1    -0.000, E3 +33656.569}
SPL {X  -165.650, Y  +383.262, Z    +0.000, E1    -6.645, E3 +33656.099}
SPL {X  -165.650, Y  +388.390, Z    +0.000, E1   -21.508, E3 +33655.886}
SPL {X  -165.650, Y  +393.439, Z    +0.000, E1   -35.398, E3 +33655.454}
SPL {X  -165.650, Y  +400.610, Z    +0.000, E1   -50.510, E3 +33655.192}
SPL {X  -165.650, Y  +414.376, Z    +0.000, E1   -68.098, E3 +33653.225}
SPL {X  -165.650, Y  +468.582, Z    +0.000, E1   -78.237, E3 +33661.995}
SPL {X  -158.306, Y  +724.277, Z    +0.000, E1   -77.461, E3 +33752.437}
ENDSPLINE

SPLINE
SPL {X  -160.145, Y  +717.851, Z    +0.000, E1   -75.386, E3 +33772.950}
ENDSPLINE

SPLINE
SPL {X  -157.156, Y  +727.862, Z    +0.000, E1   -75.175, E3 +33780.422}
SPL {X  -154.068, Y  +736.353, Z    +0.000, E1   -74.906, E3 +33787.597}
SPL {X  -149.738, Y  +746.340, Z    +0.000, E1   -74.451, E3 +33797.284}
SPL {X  -144.163, Y  +757.090, Z    +0.000, E1   -74.033, E3 +33806.377}
SPL {X  -140.473, Y  +763.291, Z    +0.000, E1   -73.478, E3 +33813.818}
SPL {X  -135.914, Y  +770.196, Z    +0.000, E1   -72.974, E3 +33820.995}
SPL {X  -131.459, Y  +776.289, Z    +0.000, E1   -72.475, E3 +33827.070}
SPL {X  -128.771, Y  +779.702, Z    +0.000, E1   -71.875, E3 +33832.017}
SPL {X  -124.506, Y  +784.762, Z    +0.000, E1   -71.815, E3 +33834.906}
SPL {X  -112.958, Y  +796.663, Z    +0.000, E1   -74.119, E3 +33831.609}
SPL {X   -51.449, Y  +832.958, Z    +0.000, E1   -57.230, E3 +33990.936}
ENDSPLINE

SPLINE
SPL {X  -123.821, Y  +785.537, Z    +0.000, E1   -64.536, E3 +34192.681}
SPL {X  -153.467, Y  +737.853, Z    +0.000, E1   -51.757, E3 +34194.996}
SPL {X  -162.176, Y  +709.248, Z    +0.000, E1   -35.773, E3 +34194.022}
SPL {X  -164.888, Y  +691.368, Z    +0.000, E1   -20.174, E3 +34192.459}
SPL {X  -165.597, Y  +679.703, Z    +0.000, E1    -7.645, E3 +34192.634}
SPL {X  -165.650, Y  +673.520, Z    +0.000, E1    -0.048, E3 +34191.586}
SPL {X  -165.650, Y  +671.692, Z    +0.000, E1    +4.450, E3 +34191.153}
SPL {X  -165.650, Y  +667.743, Z    +0.000, E1   +15.617, E3 +34191.070}
SPL {X  -165.650, Y  +661.459, Z    +0.000, E1   +33.218, E3 +34190.651}
SPL {X  -165.650, Y  +650.834, Z    +0.000, E1   +55.143, E3 +34190.039}
SPL {X  -165.650, Y  +639.785, Z    +0.000, E1   +67.512, E3 +34189.256}
SPL {X  -165.650, Y  +619.979, Z    +0.000, E1   +79.465, E3 +34185.425}
SPL {X  -165.650, Y  +569.632, Z    +0.000, E1   +78.783, E3 +34200.704}
SPL {X  -158.840, Y  +331.491, Z    +0.000, E1   +77.462, E3 +34287.014}
ENDSPLINE

SPLINE
SPL {X  -159.893, Y  +335.208, Z    +0.000, E1   +75.483, E3 +34307.748}
ENDSPLINE

SPLINE
SPL {X  -156.487, Y  +324.170, Z    +0.000, E1   +75.150, E3 +34317.130}
SPL {X  -142.256, Y  +293.629, Z    +0.000, E1   +77.020, E3 +34312.229}
ENDSPLINE

SPLINE
SPL {X  -142.811, Y  +294.566, Z    +0.000, E1   +75.668, E3 +34324.192}
ENDSPLINE

SPLINE
SPL {X  -141.646, Y  +292.615, Z    +0.000, E1   +74.702, E3 +34333.285}
SPL {X  -140.419, Y  +290.622, Z    +0.000, E1   +73.705, E3 +34342.129}
SPL {X  -136.008, Y  +283.940, Z    +0.000, E1   +73.594, E3 +34346.248}
SPL {X  -132.748, Y  +279.415, Z    +0.000, E1   +73.006, E3 +34352.303}
SPL {X  -129.007, Y  +274.590, Z    +0.000, E1   +72.484, E3 +34357.652}
SPL {X  -125.914, Y  +270.864, Z    +0.000, E1   +72.144, E3 +34361.144}
SPL {X  -123.729, Y  +268.359, Z    +0.000, E1   +71.932, E3 +34363.316}
SPL {X  -111.023, Y  +255.562, Z    +0.000, E1   +75.772, E3 +34354.182}
SPL {X   -49.289, Y  +220.353, Z    +0.000, E1   +56.690, E3 +34546.897}
ENDSPLINE

SPLINE
SPL {X  -127.117, Y  +272.287, Z    +0.000, E1   +62.713, E3 +34716.119}
SPL {X  -154.956, Y  +319.945, Z    +0.000, E1   +49.402, E3 +34720.518}
SPL {X  -162.871, Y  +348.286, Z    +0.000, E1   +32.462, E3 +34719.546}
SPL {X  -165.127, Y  +365.342, Z    +0.000, E1   +17.250, E3 +34719.384}
SPL {X  -165.640, Y  +376.693, Z    +0.000, E1    +4.721, E3 +34718.957}
SPL {X  -165.650, Y  +380.500, Z    +0.000, E1    -0.000, E3 +34718.108}
SPL {X  -165.650, Y  +383.262, Z    +0.000, E1    -6.645, E3 +34717.637}
SPL {X  -165.650, Y  +388.390, Z    +0.000, E1   -21.508, E3 +34717.425}
SPL {X  -165.650, Y  +393.439, Z    +0.000, E1   -35.398, E3 +34716.992}
SPL {X  -165.650, Y  +400.610, Z    +0.000, E1   -50.510, E3 +34716.730}
SPL {X  -165.650, Y  +414.376, Z    +0.000, E1   -68.098, E3 +34714.764}
SPL {X  -165.650, Y  +468.582, Z    +0.000, E1   -78.237, E3 +34723.534}
SPL {X  -158.306, Y  +724.277, Z    +0.000, E1   -77.461, E3 +34813.975}
ENDSPLINE

SPLINE
SPL {X  -160.145, Y  +717.851, Z    +0.000, E1   -75.386, E3 +34834.488}
ENDSPLINE

SPLINE
SPL {X  -157.156, Y  +727.862, Z    +0.000, E1   -75.175, E3 +34841.961}
SPL {X  -152.814, Y  +739.436, Z    +0.000, E1   -74.813, E3 +34851.814}
SPL {X  -148.754, Y  +748.385, Z    +0.000, E1   -74.281, E3 +34861.256}
SPL {X  -144.163, Y  +757.090, Z    +0.000, E1   -74.033, E3 +34867.915}
SPL {X  -140.473, Y  +763.291, Z    +0.000, E1   -73.478, E3 +34875.357}
SPL {X  -135.914, Y  +770.196, Z    +0.000, E1   -72.974, E3 +34882.533}
SPL {X  -131.459, Y  +776.289, Z    +0.000, E1   -72.475, E3 +34888.609}
SPL {X  -128.771, Y  +779.702, Z    +0.000, E1   -71.875, E3 +34893.556}
SPL {X  -125.267, Y  +783.889, Z    +0.000, E1   -71.674, E3 +34896.668}
SPL {X  -119.086, Y  +790.645, Z    +0.000, E1   -72.931, E3 +34894.955}
SPL {X   -51.449, Y  +832.958, Z    +0.000, E1   -57.230, E3 +35052.475}
ENDSPLINE

SPLINE
SPL {X  -113.713, Y  +795.955, Z    +0.000, E1   -65.735, E3 +35251.393}
SPL {X  -131.116, Y  +776.736, Z    +0.000, E1   -63.149, E3 +35255.923}
SPL {X  -153.467, Y  +737.853, Z    +0.000, E1   -51.757, E3 +35256.534}
SPL {X  -161.000, Y  +714.475, Z    +0.000, E1   -39.424, E3 +35256.007}
SPL {X  -164.534, Y  +694.695, Z    +0.000, E1   -23.511, E3 +35254.297}
SPL {X  -165.597, Y  +679.703, Z    +0.000, E1    -7.645, E3 +35254.173}
SPL {X  -165.650, Y  +673.520, Z    +0.000, E1    -0.048, E3 +35253.124}
SPL {X  -165.650, Y  +671.692, Z    +0.000, E1    +4.450, E3 +35252.691}
SPL {X  -165.650, Y  +667.743, Z    +0.000, E1   +15.617, E3 +35252.609}
SPL {X  -165.650, Y  +661.459, Z    +0.000, E1   +33.218, E3 +35252.189}
SPL {X  -165.650, Y  +653.296, Z    +0.000, E1   +51.333, E3 +35251.745}
SPL {X  -165.650, Y  +642.000, Z    +0.000, E1   +65.561, E3 +35250.957}
SPL {X  -165.650, Y  +619.979, Z    +0.000, E1   +79.465, E3 +35246.963}
SPL {X  -165.650, Y  +584.722, Z    +0.000, E1   +79.551, E3 +35256.254}
SPL {X  -165.650, Y  +560.326, Z    +0.000, E1   +78.360, E3 +35265.977}
SPL {X  -160.258, Y  +336.579, Z    +0.000, E1   +78.314, E3 +35337.498}
SPL {X  -159.618, Y  +334.207, Z    +0.000, E1   +75.622, E3 +35368.312}
SPL {X  -157.855, Y  +328.284, Z    +0.000, E1   +75.167, E3 +35376.278}
SPL {X  -155.139, Y  +320.432, Z    +0.000, E1   +75.106, E3 +35380.954}
SPL {X  -142.256, Y  +293.629, Z    +0.000, E1   +77.020, E3 +35373.768}
ENDSPLINE

SPLINE
SPL {X  -142.811, Y  +294.566, Z    +0.000, E1   +75.668, E3 +35385.730}
ENDSPLINE

SPLINE
SPL {X  -141.646, Y  +292.615, Z    +0.000, E1   +74.702, E3 +35394.824}
SPL {X  -140.419, Y  +290.622, Z    +0.000, E1   +73.705, E3 +35403.667}
SPL {X  -136.008, Y  +283.940, Z    +0.000, E1   +73.594, E3 +35407.786}
SPL {X  -131.988, Y  +278.404, Z    +0.000, E1   +72.860, E3 +35415.341}
SPL {X  -126.848, Y  +271.966, Z    +0.000, E1   +72.322, E3 +35421.386}
SPL {X  -123.729, Y  +268.359, Z    +0.000, E1   +71.932, E3 +35424.855}
SPL {X  -111.023, Y  +255.562, Z    +0.000, E1   +75.772, E3 +35415.720}
SPL {X   -49.289, Y  +220.353, Z    +0.000, E1   +56.690, E3 +35608.435}
ENDSPLINE

SPLINE
SPL {X  -127.117, Y  +272.287, Z    +0.000, E1   +62.713, E3 +35777.657}
SPL {X  -152.442, Y  +313.682, Z    +0.000, E1   +51.943, E3 +35781.889}
SPL {X  -162.319, Y  +345.447, Z    +0.000, E1   +34.671, E3 +35781.315}
SPL {X  -165.127, Y  +365.342, Z    +0.000, E1   +17.250, E3 +35780.923}
SPL {X  -165.640, Y  +376.693, Z    +0.000, E1    +4.721, E3 +35780.496}
SPL {X  -165.650, Y  +380.500, Z    +0.000, E1    -0.000, E3 +35779.646}
SPL {X  -165.650, Y  +383.262, Z    +0.000, E1    -6.645, E3 +35779.176}
SPL {X  -165.650, Y  +388.390, Z    +0.000, E1   -21.508, E3 +35778.963}
SPL {X  -165.650, Y  +393.439, Z    +0.000, E1   -35.398, E3 +35778.531}
SPL {X  -165.650, Y  +400.610, Z    +0.000, E1   -50.510, E3 +35778.268}
SPL {X  -165.650, Y  +414.376, Z    +0.000, E1   -68.098, E3 +35776.302}
SPL {X  -165.650, Y  +468.582, Z    +0.000, E1   -78.237, E3 +35785.072}
SPL {X  -158.306, Y  +724.277, Z    +0.000, E1   -77.461, E3 +35875.514}
ENDSPLINE

SPLINE
SPL {X  -160.145, Y  +717.851, Z    +0.000, E1   -75.386, E3 +35896.027}
ENDSPLINE

SPLINE
SPL {X  -157.156, Y  +727.862, Z    +0.000, E1   -75.175, E3 +35903.499}
SPL {X  -152.814, Y  +739.436, Z    +0.000, E1   -74.813, E3 +35913.353}
SPL {X  -147.104, Y  +751.659, Z    +0.000, E1   -74.255, E3 +35924.797}
SPL {X  -141.453, Y  +761.704, Z    +0.000, E1   -73.638, E3 +35935.010}
SPL {X  -135.914, Y  +770.196, Z    +0.000, E1   -72.974, E3 +35944.072}
SPL {X  -131.459, Y  +776.289, Z    +0.000, E1   -72.475, E3 +35950.147}
SPL {X  -127.605, Y  +781.126, Z    +0.000, E1   -71.922, E3 +35955.592}
SPL {X  -124.773, Y  +784.457, Z    +0.000, E1   -71.383, E3 +35959.639}
SPL {X  -119.086, Y  +790.645, Z    +0.000, E1   -72.931, E3 +35956.493}
SPL {X   -51.449, Y  +832.958, Z    +0.000, E1   -57.230, E3 +36114.013}
ENDSPLINE

SPLINE
SPL {X  -123.821, Y  +785.537, Z    +0.000, E1   -64.536, E3 +36315.758}
SPL {X  -153.467, Y  +737.853, Z    +0.000, E1   -51.757, E3 +36318.073}
SPL {X  -162.176, Y  +709.248, Z    +0.000, E1   -35.773, E3 +36317.098}
SPL {X  -164.888, Y  +691.368, Z    +0.000, E1   -20.174, E3 +36315.536}
SPL {X  -165.597, Y  +679.703, Z    +0.000, E1    -7.645, E3 +36315.711}
SPL {X  -165.650, Y  +673.520, Z    +0.000, E1    -0.048, E3 +36314.663}
SPL {X  -165.650, Y  +671.692, Z    +0.000, E1    +4.450, E3 +36314.230}
SPL {X  -165.650, Y  +667.743, Z    +0.000, E1   +15.617, E3 +36314.147}
SPL {X  -165.650, Y  +661.459, Z    +0.000, E1   +33.218, E3 +36313.728}
SPL {X  -165.650, Y  +653.296, Z    +0.000, E1   +51.333, E3 +36313.283}
SPL {X  -165.650, Y  +642.000, Z    +0.000, E1   +65.561, E3 +36312.495}
SPL {X  -165.650, Y  +619.979, Z    +0.000, E1   +79.465, E3 +36308.502}
SPL {X  -165.650, Y  +584.722, Z    +0.000, E1   +79.551, E3 +36317.793}
SPL {X  -165.650, Y  +560.326, Z    +0.000, E1   +78.360, E3 +36327.515}
SPL {X  -158.840, Y  +331.491, Z    +0.000, E1   +77.462, E3 +36410.091}
ENDSPLINE

SPLINE
SPL {X  -159.893, Y  +335.208, Z    +0.000, E1   +75.483, E3 +36430.825}
ENDSPLINE

SPLINE
SPL {X  -156.487, Y  +324.170, Z    +0.000, E1   +75.150, E3 +36440.207}
SPL {X  -142.256, Y  +293.629, Z    +0.000, E1   +77.020, E3 +36435.306}
ENDSPLINE

SPLINE
SPL {X  -142.811, Y  +294.566, Z    +0.000, E1   +75.668, E3 +36447.269}
ENDSPLINE

SPLINE
SPL {X  -141.646, Y  +292.615, Z    +0.000, E1   +74.702, E3 +36456.362}
SPL {X  -140.419, Y  +290.622, Z    +0.000, E1   +73.705, E3 +36465.205}
SPL {X  -136.008, Y  +283.940, Z    +0.000, E1   +73.594, E3 +36469.325}
SPL {X  -132.748, Y  +279.415, Z    +0.000, E1   +73.006, E3 +36475.380}
SPL {X  -129.007, Y  +274.590, Z    +0.000, E1   +72.484, E3 +36480.729}
SPL {X  -124.646, Y  +269.397, Z    +0.000, E1   +72.041, E3 +36485.477}
SPL {X  -111.023, Y  +255.562, Z    +0.000, E1   +75.772, E3 +36477.259}
SPL {X   -52.752, Y  +221.474, Z    +0.000, E1   +59.157, E3 +36606.511}
SPL {X   -49.901, Y  +220.545, Z    +0.000, E1   +56.696, E3 +36692.903}
ENDSPLINE

SPLINE
SPL {X  -127.117, Y  +272.287, Z    +0.000, E1   +62.713, E3 +36839.196}
SPL {X  -152.442, Y  +313.682, Z    +0.000, E1   +51.943, E3 +36843.428}
SPL {X  -159.925, Y  +335.326, Z    +0.000, E1   +41.361, E3 +36843.370}
SPL {X  -163.450, Y  +351.595, Z    +0.000, E1   +29.785, E3 +36842.481}
SPL {X  -165.127, Y  +365.342, Z    +0.000, E1   +17.250, E3 +36842.461}
SPL {X  -165.640, Y  +376.693, Z    +0.000, E1    +4.721, E3 +36842.034}
SPL {X  -165.650, Y  +380.500, Z    +0.000, E1    -0.000, E3 +36841.185}
SPL {X  -165.650, Y  +383.262, Z    +0.000, E1    -6.645, E3 +36840.714}
SPL {X  -165.650, Y  +388.390, Z    +0.000, E1   -21.508, E3 +36840.502}
SPL {X  -165.650, Y  +393.439, Z    +0.000, E1   -35.398, E3 +36840.069}
SPL {X  -165.650, Y  +400.610, Z    +0.000, E1   -50.510, E3 +36839.807}
SPL {X  -165.650, Y  +414.376, Z    +0.000, E1   -68.098, E3 +36837.841}
SPL {X  -165.650, Y  +468.582, Z    +0.000, E1   -78.237, E3 +36846.611}
SPL {X  -158.306, Y  +724.277, Z    +0.000, E1   -77.461, E3 +36937.052}
ENDSPLINE

SPLINE
SPL {X  -160.145, Y  +717.851, Z    +0.000, E1   -75.386, E3 +36957.565}
ENDSPLINE

SPLINE
SPL {X  -157.156, Y  +727.862, Z    +0.000, E1   -75.175, E3 +36965.038}
SPL {X  -154.068, Y  +736.353, Z    +0.000, E1   -74.906, E3 +36972.212}
SPL {X  -149.738, Y  +746.340, Z    +0.000, E1   -74.451, E3 +36981.900}
SPL {X  -145.204, Y  +755.223, Z    +0.000, E1   -74.188, E3 +36988.626}
SPL {X  -142.724, Y  +759.583, Z    +0.000, E1   -73.634, E3 +36995.446}
SPL {X  -138.277, Y  +766.711, Z    +0.000, E1   -73.303, E3 +37001.576}
SPL {X  -134.662, Y  +771.969, Z    +0.000, E1   -72.884, E3 +37007.019}
SPL {X  -131.459, Y  +776.289, Z    +0.000, E1   -72.475, E3 +37011.686}
SPL {X  -128.771, Y  +779.702, Z    +0.000, E1   -71.875, E3 +37016.632}
SPL {X  -125.267, Y  +783.889, Z    +0.000, E1   -71.674, E3 +37019.745}
SPL {X  -119.086, Y  +790.645, Z    +0.000, E1   -72.931, E3 +37018.032}
SPL {X   -51.449, Y  +832.958, Z    +0.000, E1   -57.230, E3 +37175.551}
ENDSPLINE

SPLINE
SPL {X  -123.821, Y  +785.537, Z    +0.000, E1   -64.536, E3 +37377.297}
SPL {X  -153.467, Y  +737.853, Z    +0.000, E1   -51.757, E3 +37379.611}
SPL {X  -162.176, Y  +709.248, Z    +0.000, E1   -35.773, E3 +37378.637}
SPL {X  -164.888, Y  +691.368, Z    +0.000, E1   -20.174, E3 +37377.075}
SPL {X  -165.597, Y  +679.703, Z    +0.000, E1    -7.645, E3 +37377.250}
SPL {X  -165.650, Y  +673.520, Z    +0.000, E1    -0.048, E3 +37376.201}
SPL {X  -165.650, Y  +671.692, Z    +0.000, E1    +4.450, E3 +37375.768}
SPL {X  -165.650, Y  +667.743, Z    +0.000, E1   +15.617, E3 +37375.686}
SPL {X  -165.650, Y  +662.891, Z    +0.000, E1   +29.740, E3 +37375.204}
SPL {X  -165.650, Y  +655.319, Z    +0.000, E1   +47.265, E3 +37375.053}
SPL {X  -165.650, Y  +642.000, Z    +0.000, E1   +65.561, E3 +37374.034}
SPL {X  -165.650, Y  +619.979, Z    +0.000, E1   +79.465, E3 +37370.040}
SPL {X  -165.650, Y  +569.632, Z    +0.000, E1   +78.783, E3 +37385.319}
SPL {X  -160.258, Y  +336.579, Z    +0.000, E1   +78.314, E3 +37460.575}
SPL {X  -159.618, Y  +334.207, Z    +0.000, E1   +75.622, E3 +37491.389}
SPL {X  -156.487, Y  +324.170, Z    +0.000, E1   +75.150, E3 +37501.745}
SPL {X  -142.256, Y  +293.629, Z    +0.000, E1   +77.020, E3 +37496.845}
ENDSPLINE

SPLINE
SPL {X  -142.811, Y  +294.566, Z    +0.000, E1   +75.668, E3 +37508.807}
ENDSPLINE

SPLINE
SPL {X  -141.646, Y  +292.615, Z    +0.000, E1   +74.702, E3 +37517.901}
SPL {X  -140.419, Y  +290.622, Z    +0.000, E1   +73.705, E3 +37526.744}
SPL {X  -136.008, Y  +283.940, Z    +0.000, E1   +73.594, E3 +37530.863}
SPL {X  -132.748, Y  +279.415, Z    +0.000, E1   +73.006, E3 +37536.919}
SPL {X  -129.007, Y  +274.590, Z    +0.000, E1   +72.484, E3 +37542.268}
SPL {X  -125.914, Y  +270.864, Z    +0.000, E1   +72.144, E3 +37545.759}
SPL {X  -123.729, Y  +268.359, Z    +0.000, E1   +71.932, E3 +37547.932}
SPL {X  -111.023, Y  +255.562, Z    +0.000, E1   +75.772, E3 +37538.797}
SPL {X   -49.289, Y  +220.353, Z    +0.000, E1   +56.690, E3 +37731.512}
ENDSPLINE

SPLINE
SPL {X  -127.117, Y  +272.287, Z    +0.000, E1   +62.713, E3 +37900.734}
SPL {X  -152.442, Y  +313.682, Z    +0.000, E1   +51.943, E3 +37904.966}
SPL {X  -159.925, Y  +335.326, Z    +0.000, E1   +41.361, E3 +37904.908}
SPL {X  -163.450, Y  +351.595, Z    +0.000, E1   +29.785, E3 +37904.019}
SPL {X  -165.127, Y  +365.342, Z    +0.000, E1   +17.250, E3 +37904.000}
SPL {X  -165.640, Y  +376.693, Z    +0.000, E1    +4.721, E3 +37903.572}
SPL {X  -165.650, Y  +380.500, Z    +0.000, E1    -0.000, E3 +37902.723}
SPL {X  -165.650, Y  +382.123, Z    +0.000, E1    -3.912, E3 +37902.351}
SPL {X  -165.650, Y  +387.069, Z    +0.000, E1   -17.420, E3 +37902.062}
SPL {X  -165.650, Y  +393.439, Z    +0.000, E1   -35.398, E3 +37901.608}
SPL {X  -165.650, Y  +400.610, Z    +0.000, E1   -50.510, E3 +37901.345}
SPL {X  -165.650, Y  +414.376, Z    +0.000, E1   -68.098, E3 +37899.379}
SPL {X  -165.650, Y  +468.582, Z    +0.000, E1   -78.237, E3 +37908.149}
SPL {X  -160.244, Y  +717.475, Z    +0.000, E1   -78.917, E3 +37980.707}
SPL {X  -159.651, Y  +719.676, Z    +0.000, E1   -75.661, E3 +38017.094}
SPL {X  -157.156, Y  +727.862, Z    +0.000, E1   -75.175, E3 +38026.576}
SPL {X  -152.814, Y  +739.436, Z    +0.000, E1   -74.813, E3 +38036.430}
SPL {X  -148.754, Y  +748.385, Z    +0.000, E1   -74.281, E3 +38045.872}
SPL {X  -144.163, Y  +757.090, Z    +0.000, E1   -74.033, E3 +38052.531}
SPL {X  -139.284, Y  +765.165, Z    +0.000, E1   -73.322, E3 +38062.225}
SPL {X  -134.662, Y  +771.969, Z    +0.000, E1   -72.884, E3 +38068.557}
SPL {X  -131.459, Y  +776.289, Z    +0.000, E1   -72.475, E3 +38073.224}
SPL {X  -128.771, Y  +779.702, Z    +0.000, E1   -71.875, E3 +38078.171}
SPL {X  -124.506, Y  +784.762, Z    +0.000, E1   -71.815, E3 +38081.059}
SPL {X  -112.958, Y  +796.663, Z    +0.000, E1   -74.119, E3 +38077.763}
SPL {X   -54.274, Y  +832.006, Z    +0.000, E1   -58.502, E3 +38209.783}
SPL {X   -50.797, Y  +833.169, Z    +0.000, E1   -57.000, E3 +38305.132}
ENDSPLINE

SPLINE
SPL {X  -113.713, Y  +795.955, Z    +0.000, E1   -65.735, E3 +38436.008}
SPL {X  -131.116, Y  +776.736, Z    +0.000, E1   -63.149, E3 +38440.538}
SPL {X  -153.467, Y  +737.853, Z    +0.000, E1   -51.757, E3 +38441.150}
SPL {X  -162.176, Y  +709.248, Z    +0.000, E1   -35.773, E3 +38440.175}
SPL {X  -164.888, Y  +691.368, Z    +0.000, E1   -20.174, E3 +38438.613}
SPL {X  -165.597, Y  +679.703, Z    +0.000, E1    -7.645, E3 +38438.788}
SPL {X  -165.650, Y  +673.520, Z    +0.000, E1    -0.048, E3 +38437.740}
SPL {X  -165.650, Y  +671.692, Z    +0.000, E1    +4.450, E3 +38437.306}
SPL {X  -165.650, Y  +667.743, Z    +0.000, E1   +15.617, E3 +38437.224}
SPL {X  -165.650, Y  +662.891, Z    +0.000, E1   +29.740, E3 +38436.742}
SPL {X  -165.650, Y  +655.319, Z    +0.000, E1   +47.265, E3 +38436.591}
SPL {X  -165.650, Y  +642.000, Z    +0.000, E1   +65.561, E3 +38435.572}
SPL {X  -165.650, Y  +619.979, Z    +0.000, E1   +79.465, E3 +38431.579}
SPL {X  -165.650, Y  +569.632, Z    +0.000, E1   +78.783, E3 +38446.858}
SPL {X  -158.840, Y  +331.491, Z    +0.000, E1   +77.462, E3 +38533.168}
ENDSPLINE

SPLINE
SPL {X  -159.893, Y  +335.208, Z    +0.000, E1   +75.483, E3 +38553.902}
ENDSPLINE

SPLINE
SPL {X  -156.487, Y  +324.170, Z    +0.000, E1   +75.150, E3 +38563.283}
SPL {X  -142.256, Y  +293.629, Z    +0.000, E1   +77.020, E3 +38558.383}
ENDSPLINE

SPLINE
SPL {X  -142.811, Y  +294.566, Z    +0.000, E1   +75.668, E3 +38570.346}
ENDSPLINE

SPLINE
SPL {X  -141.646, Y  +292.615, Z    +0.000, E1   +74.702, E3 +38579.439}
SPL {X  -140.419, Y  +290.622, Z    +0.000, E1   +73.705, E3 +38588.282}
SPL {X  -135.839, Y  +283.697, Z    +0.000, E1   +73.388, E3 +38594.021}
SPL {X  -131.336, Y  +277.551, Z    +0.000, E1   +72.879, E3 +38600.273}
SPL {X  -126.848, Y  +271.966, Z    +0.000, E1   +72.322, E3 +38606.001}
SPL {X  -123.729, Y  +268.359, Z    +0.000, E1   +71.932, E3 +38609.470}
SPL {X  -111.023, Y  +255.562, Z    +0.000, E1   +75.772, E3 +38600.336}
SPL {X   -52.752, Y  +221.474, Z    +0.000, E1   +59.157, E3 +38729.587}
SPL {X   -49.901, Y  +220.545, Z    +0.000, E1   +56.696, E3 +38815.980}
ENDSPLINE

SPLINE
SPL {X  -127.117, Y  +272.287, Z    +0.000, E1   +62.713, E3 +38962.273}
SPL {X  -152.442, Y  +313.682, Z    +0.000, E1   +51.943, E3 +38966.505}
SPL {X  -162.319, Y  +345.447, Z    +0.000, E1   +34.671, E3 +38965.930}
SPL {X  -165.127, Y  +365.342, Z    +0.000, E1   +17.250, E3 +38965.538}
SPL {X  -165.640, Y  +376.693, Z    +0.000, E1    +4.721, E3 +38965.111}
SPL {X  -165.650, Y  +380.500, Z    +0.000, E1    -0.000, E3 +38964.262}
SPL {X  -165.650, Y  +383.262, Z    +0.000, E1    -6.645, E3 +38963.791}
SPL {X  -165.650, Y  +388.390, Z    +0.000, E1   -21.508, E3 +38963.579}
SPL {X  -165.650, Y  +393.439, Z    +0.000, E1   -35.398, E3 +38963.146}
SPL {X  -165.650, Y  +400.610, Z    +0.000, E1   -50.510, E3 +38962.884}
SPL {X  -165.650, Y  +414.376, Z    +0.000, E1   -68.098, E3 +38960.917}
SPL {X  -165.650, Y  +468.582, Z    +0.000, E1   -78.237, E3 +38969.688}
SPL {X  -158.306, Y  +724.277, Z    +0.000, E1   -77.461, E3 +39060.129}
ENDSPLINE

SPLINE
SPL {X  -160.145, Y  +717.851, Z    +0.000, E1   -75.386, E3 +39080.642}
ENDSPLINE

SPLINE
SPL {X  -157.156, Y  +727.862, Z    +0.000, E1   -75.175, E3 +39088.114}
SPL {X  -152.814, Y  +739.436, Z    +0.000, E1   -74.813, E3 +39097.968}
SPL {X  -148.754, Y  +748.385, Z    +0.000, E1   -74.281, E3 +39107.410}
SPL {X  -144.163, Y  +757.090, Z    +0.000, E1   -74.033, E3 +39114.069}
SPL {X  -139.284, Y  +765.165, Z    +0.000, E1   -73.322, E3 +39123.764}
SPL {X  -134.662, Y  +771.969, Z    +0.000, E1   -72.884, E3 +39130.096}
SPL {X  -131.459, Y  +776.289, Z    +0.000, E1   -72.475, E3 +39134.763}
SPL {X  -127.605, Y  +781.126, Z    +0.000, E1   -71.922, E3 +39140.207}
SPL {X  -124.773, Y  +784.457, Z    +0.000, E1   -71.383, E3 +39144.254}
SPL {X  -119.086, Y  +790.645, Z    +0.000, E1   -72.931, E3 +39141.109}
SPL {X   -51.449, Y  +832.958, Z    +0.000, E1   -57.230, E3 +39298.628}
ENDSPLINE

SPLINE
SPL {X  -123.821, Y  +785.537, Z    +0.000, E1   -64.536, E3 +39500.374}
SPL {X  -153.467, Y  +737.853, Z    +0.000, E1   -51.757, E3 +39502.688}
SPL {X  -162.176, Y  +709.248, Z    +0.000, E1   -35.773, E3 +39501.714}
SPL {X  -164.888, Y  +691.368, Z    +0.000, E1   -20.174, E3 +39500.151}
SPL {X  -165.597, Y  +679.703, Z    +0.000, E1    -7.645, E3 +39500.327}
SPL {X  -165.650, Y  +673.520, Z    +0.000, E1    -0.048, E3 +39499.278}
SPL {X  -165.650, Y  +671.692, Z    +0.000, E1    +4.450, E3 +39498.845}
SPL {X  -165.650, Y  +667.743, Z    +0.000, E1   +15.617, E3 +39498.763}
SPL {X  -165.650, Y  +661.459, Z    +0.000, E1   +33.218, E3 +39498.343}
SPL {X  -165.650, Y  +653.296, Z    +0.000, E1   +51.333, E3 +39497.899}
SPL {X  -165.650, Y  +642.000, Z    +0.000, E1   +65.561, E3 +39497.111}
SPL {X  -165.650, Y  +619.979, Z    +0.000, E1   +79.465, E3 +39493.117}
SPL {X  -165.650, Y  +584.722, Z    +0.000, E1   +79.551, E3 +39502.408}
SPL {X  -165.650, Y  +560.326, Z    +0.000, E1   +78.360, E3 +39512.131}
SPL {X  -158.840, Y  +331.491, Z    +0.000, E1   +77.462, E3 +39594.706}
ENDSPLINE

SPLINE
SPL {X  -159.893, Y  +335.208, Z    +0.000, E1   +75.483, E3 +39615.441}
ENDSPLINE

SPLINE
SPL {X  -156.487, Y  +324.170, Z    +0.000, E1   +75.150, E3 +39624.822}
SPL {X  -142.256, Y  +293.629, Z    +0.000, E1   +77.020, E3 +39619.922}
ENDSPLINE

SPLINE
SPL {X  -142.811, Y  +294.566, Z    +0.000, E1   +75.668, E3 +39631.884}
ENDSPLINE

SPLINE
SPL {X  -141.646, Y  +292.615, Z    +0.000, E1   +74.702, E3 +39640.978}
SPL {X  -140.419, Y  +290.622, Z    +0.000, E1   +73.705, E3 +39649.821}
SPL {X  -136.008, Y  +283.940, Z    +0.000, E1   +73.594, E3 +39653.940}
SPL {X  -132.748, Y  +279.415, Z    +0.000, E1   +73.006, E3 +39659.996}
SPL {X  -129.007, Y  +274.590, Z    +0.000, E1   +72.484, E3 +39665.345}
SPL {X  -124.646, Y  +269.397, Z    +0.000, E1   +72.041, E3 +39670.093}
SPL {X  -111.023, Y  +255.562, Z    +0.000, E1   +75.772, E3 +39661.874}
SPL {X   -52.752, Y  +221.474, Z    +0.000, E1   +59.157, E3 +39791.126}
SPL {X   -49.901, Y  +220.545, Z    +0.000, E1   +56.696, E3 +39877.518}
ENDSPLINE

SPLINE
SPL {X  -127.117, Y  +272.287, Z    +0.000, E1   +62.713, E3 +40023.811}
SPL {X  -152.442, Y  +313.682, Z    +0.000, E1   +51.943, E3 +40028.043}
SPL {X  -159.925, Y  +335.326, Z    +0.000, E1   +41.361, E3 +40027.985}
SPL {X  -163.450, Y  +351.595, Z    +0.000, E1   +29.785, E3 +40027.096}
SPL {X  -165.127, Y  +365.342, Z    +0.000, E1   +17.250, E3 +40027.076}
SPL {X  -165.640, Y  +376.693, Z    +0.000, E1    +4.721, E3 +40026.649}
SPL {X  -165.650, Y  +380.500, Z    +0.000, E1    -0.000, E3 +40025.800}
SPL {X  -165.650, Y  +383.262, Z    +0.000, E1    -6.645, E3 +40025.329}
SPL {X  -165.650, Y  +388.390, Z    +0.000, E1   -21.508, E3 +40025.117}
SPL {X  -165.650, Y  +393.439, Z    +0.000, E1   -35.398, E3 +40024.685}
SPL {X  -165.650, Y  +400.610, Z    +0.000, E1   -50.510, E3 +40024.422}
SPL {X  -165.650, Y  +414.376, Z    +0.000, E1   -68.098, E3 +40022.456}
SPL {X  -165.650, Y  +468.582, Z    +0.000, E1   -78.237, E3 +40031.226}
SPL {X  -158.306, Y  +724.277, Z    +0.000, E1   -77.461, E3 +40121.667}
ENDSPLINE

SPLINE
SPL {X  -160.145, Y  +717.851, Z    +0.000, E1   -75.386, E3 +40142.181}
ENDSPLINE

SPLINE
SPL {X  -157.156, Y  +727.862, Z    +0.000, E1   -75.175, E3 +40149.653}
SPL {X  -152.814, Y  +739.436, Z    +0.000, E1   -74.813, E3 +40159.507}
SPL {X  -147.104, Y  +751.659, Z    +0.000, E1   -74.255, E3 +40170.951}
SPL {X  -141.453, Y  +761.704, Z    +0.000, E1   -73.638, E3 +40181.164}
SPL {X  -135.914, Y  +770.196, Z    +0.000, E1   -72.974, E3 +40190.225}
SPL {X  -131.459, Y  +776.289, Z    +0.000, E1   -72.475, E3 +40196.301}
SPL {X  -127.605, Y  +781.126, Z    +0.000, E1   -71.922, E3 +40201.745}
SPL {X  -124.773, Y  +784.457, Z    +0.000, E1   -71.383, E3 +40205.793}
SPL {X  -119.086, Y  +790.645, Z    +0.000, E1   -72.931, E3 +40202.647}
SPL {X   -51.449, Y  +832.958, Z    +0.000, E1   -57.230, E3 +40360.167}
ENDSPLINE

SPLINE
SPL {X  -113.713, Y  +795.955, Z    +0.000, E1   -65.735, E3 +40559.085}
SPL {X  -131.116, Y  +776.736, Z    +0.000, E1   -63.149, E3 +40563.615}
SPL {X  -153.467, Y  +737.853, Z    +0.000, E1   -51.757, E3 +40564.227}
SPL {X  -161.000, Y  +714.475, Z    +0.000, E1   -39.424, E3 +40563.699}
SPL {X  -164.534, Y  +694.695, Z    +0.000, E1   -23.511, E3 +40561.989}
SPL {X  -165.597, Y  +679.703, Z    +0.000, E1    -7.645, E3 +40561.865}
SPL {X  -165.650, Y  +673.520, Z    +0.000, E1    -0.048, E3 +40560.817}
SPL {X  -165.650, Y  +671.692, Z    +0.000, E1    +4.450, E3 +40560.383}
SPL {X  -165.650, Y  +667.743, Z    +0.000, E1   +15.617, E3 +40560.301}
SPL {X  -165.650, Y  +661.459, Z    +0.000, E1   +33.218, E3 +40559.882}
SPL {X  -165.650, Y  +650.834, Z    +0.000, E1   +55.143, E3 +40559.270}
SPL {X  -165.650, Y  +639.785, Z    +0.000, E1   +67.512, E3 +40558.487}
SPL {X  -165.650, Y  +619.979, Z    +0.000, E1   +79.465, E3 +40554.656}
SPL {X  -165.650, Y  +584.722, Z    +0.000, E1   +79.551, E3 +40563.947}
SPL {X  -165.650, Y  +560.326, Z    +0.000, E1   +78.360, E3 +40573.669}
SPL {X  -160.258, Y  +336.579, Z    +0.000, E1   +78.314, E3 +40645.191}
SPL {X  -159.618, Y  +334.207, Z    +0.000, E1   +75.622, E3 +40676.005}
SPL {X  -156.487, Y  +324.170, Z    +0.000, E1   +75.150, E3 +40686.360}
SPL {X  -142.256, Y  +293.629, Z    +0.000, E1   +77.020, E3 +40681.460}
ENDSPLINE

SPLINE
SPL {X  -142.811, Y  +294.566, Z    +0.000, E1   +75.668, E3 +40693.422}
ENDSPLINE

SPLINE
SPL {X  -141.646, Y  +292.615, Z    +0.000, E1   +74.702, E3 +40702.516}
SPL {X  -140.419, Y  +290.622, Z    +0.000, E1   +73.705, E3 +40711.359}
SPL {X  -135.839, Y  +283.697, Z    +0.000, E1   +73.388, E3 +40717.097}
SPL {X  -131.903, Y  +278.292, Z    +0.000, E1   +73.096, E3 +40721.587}
SPL {X  -129.007, Y  +274.590, Z    +0.000, E1   +72.484, E3 +40726.883}
SPL {X  -124.646, Y  +269.397, Z    +0.000, E1   +72.041, E3 +40731.631}
SPL {X  -111.023, Y  +255.562, Z    +0.000, E1   +75.772, E3 +40723.413}
SPL {X   -49.289, Y  +220.353, Z    +0.000, E1   +56.690, E3 +40916.128}
ENDSPLINE

SPLINE
SPL {X  -127.117, Y  +272.287, Z    +0.000, E1   +62.713, E3 +41085.350}
SPL {X  -152.442, Y  +313.682, Z    +0.000, E1   +51.943, E3 +41089.581}
SPL {X  -159.925, Y  +335.326, Z    +0.000, E1   +41.361, E3 +41089.523}
SPL {X  -163.450, Y  +351.595, Z    +0.000, E1   +29.785, E3 +41088.635}
SPL {X  -165.127, Y  +365.342, Z    +0.000, E1   +17.250, E3 +41088.615}
SPL {X  -165.640, Y  +376.693, Z    +0.000, E1    +4.721, E3 +41088.188}
SPL {X  -165.650, Y  +380.500, Z    +0.000, E1    -0.000, E3 +41087.339}
SPL {X  -165.650, Y  +382.123, Z    +0.000, E1    -3.912, E3 +41086.966}
SPL {X  -165.650, Y  +387.069, Z    +0.000, E1   -17.420, E3 +41086.677}
SPL {X  -165.650, Y  +393.439, Z    +0.000, E1   -35.398, E3 +41086.223}
SPL {X  -165.650, Y  +402.896, Z    +0.000, E1   -54.480, E3 +41085.464}
SPL {X  -165.650, Y  +416.934, Z    +0.000, E1   -69.887, E3 +41083.930}
SPL {X  -165.650, Y  +459.729, Z    +0.000, E1   -78.035, E3 +41090.449}
SPL {X  -165.650, Y  +475.450, Z    +0.000, E1   -78.345, E3 +41094.563}
SPL {X  -160.244, Y  +717.475, Z    +0.000, E1   -78.917, E3 +41165.322}
SPL {X  -159.651, Y  +719.676, Z    +0.000, E1   -75.661, E3 +41201.709}
SPL {X  -157.156, Y  +727.862, Z    +0.000, E1   -75.175, E3 +41211.191}
SPL {X  -152.814, Y  +739.436, Z    +0.000, E1   -74.813, E3 +41221.045}
SPL {X  -148.754, Y  +748.385, Z    +0.000, E1   -74.281, E3 +41230.487}
SPL {X  -144.163, Y  +757.090, Z    +0.000, E1   -74.033, E3 +41237.146}
SPL {X  -140.473, Y  +763.291, Z    +0.000, E1   -73.478, E3 +41244.588}
SPL {X  -135.914, Y  +770.196, Z    +0.000, E1   -72.974, E3 +41251.764}
SPL {X  -131.459, Y  +776.289, Z    +0.000, E1   -72.475, E3 +41257.840}
SPL {X  -128.771, Y  +779.702, Z    +0.000, E1   -71.875, E3 +41262.786}
SPL {X  -124.506, Y  +784.762, Z    +0.000, E1   -71.815, E3 +41265.675}
SPL {X  -112.958, Y  +796.663, Z    +0.000, E1   -74.119, E3 +41262.378}
SPL {X   -51.449, Y  +832.958, Z    +0.000, E1   -57.230, E3 +41421.705}
ENDSPLINE

SPLINE
SPL {X  -123.821, Y  +785.537, Z    +0.000, E1   -64.536, E3 +41623.450}
SPL {X  -153.467, Y  +737.853, Z    +0.000, E1   -51.757, E3 +41625.765}
SPL {X  -161.000, Y  +714.475, Z    +0.000, E1   -39.424, E3 +41625.238}
SPL {X  -164.534, Y  +694.695, Z    +0.000, E1   -23.511, E3 +41623.528}
SPL {X  -165.597, Y  +679.703, Z    +0.000, E1    -7.645, E3 +41623.403}
SPL {X  -165.650, Y  +673.520, Z    +0.000, E1    -0.048, E3 +41622.355}
SPL {X  -165.650, Y  +671.692, Z    +0.000, E1    +4.450, E3 +41621.922}
SPL {X  -165.650, Y  +667.743, Z    +0.000, E1   +15.617, E3 +41621.840}
SPL {X  -165.650, Y  +662.891, Z    +0.000, E1   +29.740, E3 +41621.358}
SPL {X  -165.650, Y  +655.319, Z    +0.000, E1   +47.265, E3 +41621.206}
SPL {X  -165.650, Y  +642.000, Z    +0.000, E1   +65.561, E3 +41620.188}
SPL {X  -165.650, Y  +619.979, Z    +0.000, E1   +79.465, E3 +41616.194}
SPL {X  -165.650, Y  +569.632, Z    +0.000, E1   +78.783, E3 +41631.473}
SPL {X  -158.840, Y  +331.491, Z    +0.000, E1   +77.462, E3 +41717.783}
ENDSPLINE

SPLINE
SPL {X  -159.893, Y  +335.208, Z    +0.000, E1   +75.483, E3 +41738.518}
ENDSPLINE

SPLINE
SPL {X  -156.487, Y  +324.170, Z    +0.000, E1   +75.150, E3 +41747.899}
SPL {X  -142.256, Y  +293.629, Z    +0.000, E1   +77.020, E3 +41742.999}
ENDSPLINE

SPLINE
SPL {X  -142.811, Y  +294.566, Z    +0.000, E1   +75.668, E3 +41754.961}
ENDSPLINE

SPLINE
SPL {X  -141.646, Y  +292.615, Z    +0.000, E1   +74.702, E3 +41764.055}
SPL {X  -140.419, Y  +290.622, Z    +0.000, E1   +73.705, E3 +41772.898}
SPL {X  -135.839, Y  +283.697, Z    +0.000, E1   +73.388, E3 +41778.636}
SPL {X  -131.336, Y  +277.551, Z    +0.000, E1   +72.879, E3 +41784.888}
SPL {X  -126.848, Y  +271.966, Z    +0.000, E1   +72.322, E3 +41790.617}
SPL {X  -123.729, Y  +268.359, Z    +0.000, E1   +71.932, E3 +41794.085}
SPL {X  -111.023, Y  +255.562, Z    +0.000, E1   +75.772, E3 +41784.951}
SPL {X   -52.752, Y  +221.474, Z    +0.000, E1   +59.157, E3 +41914.203}
SPL {X   -49.901, Y  +220.545, Z    +0.000, E1   +56.696, E3 +42000.595}
ENDSPLINE

SPLINE
SPL {X  -127.117, Y  +272.287, Z    +0.000, E1   +62.713, E3 +42146.888}
SPL {X  -152.442, Y  +313.682, Z    +0.000, E1   +51.943, E3 +42151.120}
SPL {X  -162.319, Y  +345.447, Z    +0.000, E1   +34.671, E3 +42150.545}
SPL {X  -165.127, Y  +365.342, Z    +0.000, E1   +17.250, E3 +42150.153}
SPL {X  -165.640, Y  +376.693, Z    +0.000, E1    +4.721, E3 +42149.726}
SPL {X  -165.650, Y  +380.500, Z    +0.000, E1    -0.000, E3 +42148.877}
SPL {X  -165.650, Y  +383.262, Z    +0.000, E1    -6.645, E3 +42148.406}
SPL {X  -165.650, Y  +388.390, Z    +0.000, E1   -21.508, E3 +42148.194}
SPL {X  -165.650, Y  +393.439, Z    +0.000, E1   -35.398, E3 +42147.762}
SPL {X  -165.650, Y  +400.610, Z    +0.000, E1   -50.510, E3 +42147.499}
SPL {X  -165.650, Y  +414.376, Z    +0.000, E1   -68.098, E3 +42145.533}
SPL {X  -165.650, Y  +468.582, Z    +0.000, E1   -78.237, E3 +42154.303}
SPL {X  -158.306, Y  +724.277, Z    +0.000, E1   -77.461, E3 +42244.744}
ENDSPLINE

SPLINE
SPL {X  -160.145, Y  +717.851, Z    +0.000, E1   -75.386, E3 +42265.258}
ENDSPLINE

SPLINE
SPL {X  -157.156, Y  +727.862, Z    +0.000, E1   -75.175, E3 +42272.730}
SPL {X  -152.814, Y  +739.436, Z    +0.000, E1   -74.813, E3 +42282.583}
SPL {X  -147.104, Y  +751.659, Z    +0.000, E1   -74.255, E3 +42294.028}
SPL {X  -141.453, Y  +761.704, Z    +0.000, E1   -73.638, E3 +42304.241}
SPL {X  -135.914, Y  +770.196, Z    +0.000, E1   -72.974, E3 +42313.302}
SPL {X  -131.459, Y  +776.289, Z    +0.000, E1   -72.475, E3 +42319.378}
SPL {X  -128.771, Y  +779.702, Z    +0.000, E1   -71.875, E3 +42324.325}
SPL {X  -124.506, Y  +784.762, Z    +0.000, E1   -71.815, E3 +42327.213}
SPL {X  -112.958, Y  +796.663, Z    +0.000, E1   -74.119, E3 +42323.917}
SPL {X   -54.274, Y  +832.006, Z    +0.000, E1   -58.502, E3 +42455.937}
SPL {X   -50.797, Y  +833.169, Z    +0.000, E1   -57.000, E3 +42551.286}
ENDSPLINE

SPLINE
SPL {X  -113.713, Y  +795.955, Z    +0.000, E1   -65.735, E3 +42682.162}
SPL {X  -131.116, Y  +776.736, Z    +0.000, E1   -63.149, E3 +42686.692}
SPL {X  -153.467, Y  +737.853, Z    +0.000, E1   -51.757, E3 +42687.304}
SPL {X  -162.176, Y  +709.248, Z    +0.000, E1   -35.773, E3 +42686.329}
SPL {X  -164.888, Y  +691.368, Z    +0.000, E1   -20.174, E3 +42684.767}
SPL {X  -165.597, Y  +679.703, Z    +0.000, E1    -7.645, E3 +42684.942}
SPL {X  -165.650, Y  +673.520, Z    +0.000, E1    -0.048, E3 +42683.894}
SPL {X  -165.650, Y  +671.692, Z    +0.000, E1    +4.450, E3 +42683.460}
SPL {X  -165.650, Y  +667.743, Z    +0.000, E1   +15.617, E3 +42683.378}
SPL {X  -165.650, Y  +662.891, Z    +0.000, E1   +29.740, E3 +42682.896}
SPL {X  -165.650, Y  +655.319, Z    +0.000, E1   +47.265, E3 +42682.745}
SPL {X  -165.650, Y  +642.000, Z    +0.000, E1   +65.561, E3 +42681.726}
SPL {X  -165.650, Y  +619.979, Z    +0.000, E1   +79.465, E3 +42677.733}
SPL {X  -165.650, Y  +569.632, Z    +0.000, E1   +78.783, E3 +42693.011}
SPL {X  -158.840, Y  +331.491, Z    +0.000, E1   +77.462, E3 +42779.322}
ENDSPLINE

SPLINE
SPL {X  -159.893, Y  +335.208, Z    +0.000, E1   +75.483, E3 +42800.056}
ENDSPLINE

SPLINE
SPL {X  -156.487, Y  +324.170, Z    +0.000, E1   +75.150, E3 +42809.437}
SPL {X  -142.256, Y  +293.629, Z    +0.000, E1   +77.020, E3 +42804.537}
ENDSPLINE

SPLINE
SPL {X  -142.811, Y  +294.566, Z    +0.000, E1   +75.668, E3 +42816.499}
ENDSPLINE

SPLINE
SPL {X  -141.646, Y  +292.615, Z    +0.000, E1   +74.702, E3 +42825.593}
SPL {X  -140.419, Y  +290.622, Z    +0.000, E1   +73.705, E3 +42834.436}
SPL {X  -135.839, Y  +283.697, Z    +0.000, E1   +73.388, E3 +42840.174}
SPL {X  -131.336, Y  +277.551, Z    +0.000, E1   +72.879, E3 +42846.427}
SPL {X  -126.848, Y  +271.966, Z    +0.000, E1   +72.322, E3 +42852.155}
SPL {X  -123.729, Y  +268.359, Z    +0.000, E1   +71.932, E3 +42855.624}
SPL {X  -111.023, Y  +255.562, Z    +0.000, E1   +75.772, E3 +42846.490}
SPL {X   -49.289, Y  +220.353, Z    +0.000, E1   +56.690, E3 +43039.205}
ENDSPLINE

SPLINE
SPL {X  -127.117, Y  +272.287, Z    +0.000, E1   +62.713, E3 +43208.427}
SPL {X  -154.956, Y  +319.945, Z    +0.000, E1   +49.402, E3 +43212.826}
SPL {X  -162.871, Y  +348.286, Z    +0.000, E1   +32.462, E3 +43211.853}
SPL {X  -165.127, Y  +365.342, Z    +0.000, E1   +17.250, E3 +43211.692}
SPL {X  -165.640, Y  +376.693, Z    +0.000, E1    +4.721, E3 +43211.265}
SPL {X  -165.650, Y  +380.500, Z    +0.000, E1    -0.000, E3 +43210.416}
SPL {X  -165.650, Y  +383.262, Z    +0.000, E1    -6.645, E3 +43209.945}
SPL {X  -165.650, Y  +388.390, Z    +0.000, E1   -21.508, E3 +43209.733}
SPL {X  -165.650, Y  +393.439, Z    +0.000, E1   -35.398, E3 +43209.300}
SPL {X  -165.650, Y  +400.610, Z    +0.000, E1   -50.510, E3 +43209.038}
SPL {X  -165.650, Y  +414.376, Z    +0.000, E1   -68.098, E3 +43207.071}
SPL {X  -165.650, Y  +468.582, Z    +0.000, E1   -78.237, E3 +43215.841}
SPL {X  -158.306, Y  +724.277, Z    +0.000, E1   -77.461, E3 +43306.283}
ENDSPLINE

SPLINE
SPL {X  -160.145, Y  +717.851, Z    +0.000, E1   -75.386, E3 +43326.796}
ENDSPLINE

SPLINE
SPL {X  -157.156, Y  +727.862, Z    +0.000, E1   -75.175, E3 +43334.268}
SPL {X  -154.068, Y  +736.353, Z    +0.000, E1   -74.906, E3 +43341.443}
SPL {X  -149.738, Y  +746.340, Z    +0.000, E1   -74.451, E3 +43351.131}
SPL {X  -144.163, Y  +757.090, Z    +0.000, E1   -74.033, E3 +43360.223}
SPL {X  -140.473, Y  +763.291, Z    +0.000, E1   -73.478, E3 +43367.665}
SPL {X  -135.914, Y  +770.196, Z    +0.000, E1   -72.974, E3 +43374.841}
SPL {X  -131.459, Y  +776.289, Z    +0.000, E1   -72.475, E3 +43380.917}
SPL {X  -128.771, Y  +779.702, Z    +0.000, E1   -71.875, E3 +43385.863}
SPL {X  -124.506, Y  +784.762, Z    +0.000, E1   -71.815, E3 +43388.752}
SPL {X  -112.958, Y  +796.663, Z    +0.000, E1   -74.119, E3 +43385.455}
SPL {X   -51.449, Y  +832.958, Z    +0.000, E1   -57.230, E3 +43544.782}
ENDSPLINE

SPLINE
SPL {X  -123.821, Y  +785.537, Z    +0.000, E1   -64.536, E3 +43746.527}
SPL {X  -153.467, Y  +737.853, Z    +0.000, E1   -51.757, E3 +43748.842}
SPL {X  -162.176, Y  +709.248, Z    +0.000, E1   -35.773, E3 +43747.868}
SPL {X  -164.888, Y  +691.368, Z    +0.000, E1   -20.174, E3 +43746.305}
SPL {X  -165.597, Y  +679.703, Z    +0.000, E1    -7.645, E3 +43746.480}
SPL {X  -165.650, Y  +673.520, Z    +0.000, E1    -0.048, E3 +43745.432}
SPL {X  -165.650, Y  +671.692, Z    +0.000, E1    +4.450, E3 +43744.999}
SPL {X  -165.650, Y  +667.743, Z    +0.000, E1   +15.617, E3 +43744.917}
SPL {X  -165.650, Y  +661.459, Z    +0.000, E1   +33.218, E3 +43744.497}
SPL {X  -165.650, Y  +650.834, Z    +0.000, E1   +55.143, E3 +43743.885}
SPL {X  -165.650, Y  +639.785, Z    +0.000, E1   +67.512, E3 +43743.102}
SPL {X  -165.650, Y  +619.979, Z    +0.000, E1   +79.465, E3 +43739.271}
SPL {X  -165.650, Y  +569.632, Z    +0.000, E1   +78.783, E3 +43754.550}
SPL {X  -158.840, Y  +331.491, Z    +0.000, E1   +77.462, E3 +43840.860}
ENDSPLINE

SPLINE
SPL {X  -159.893, Y  +335.208, Z    +0.000, E1   +75.483, E3 +43861.595}
ENDSPLINE

SPLINE
SPL {X  -156.487, Y  +324.170, Z    +0.000, E1   +75.150, E3 +43870.976}
SPL {X  -142.256, Y  +293.629, Z    +0.000, E1   +77.020, E3 +43866.076}
ENDSPLINE

SPLINE
SPL {X  -142.811, Y  +294.566, Z    +0.000, E1   +75.668, E3 +43878.038}
ENDSPLINE

SPLINE
SPL {X  -141.646, Y  +292.615, Z    +0.000, E1   +74.702, E3 +43887.131}
SPL {X  -140.419, Y  +290.622, Z    +0.000, E1   +73.705, E3 +43895.975}
SPL {X  -136.008, Y  +283.940, Z    +0.000, E1   +73.594, E3 +43900.094}
SPL {X  -132.748, Y  +279.415, Z    +0.000, E1   +73.006, E3 +43906.150}
SPL {X  -129.007, Y  +274.590, Z    +0.000, E1   +72.484, E3 +43911.498}
SPL {X  -125.914, Y  +270.864, Z    +0.000, E1   +72.144, E3 +43914.990}
SPL {X  -123.729, Y  +268.359, Z    +0.000, E1   +71.932, E3 +43917.162}
SPL {X  -111.023, Y  +255.562, Z    +0.000, E1   +75.772, E3 +43908.028}
SPL {X   -49.289, Y  +220.353, Z    +0.000, E1   +56.690, E3 +44100.743}
ENDSPLINE

SPLINE
SPL {X  -127.117, Y  +272.287, Z    +0.000, E1   +62.713, E3 +44269.965}
SPL {X  -154.956, Y  +319.945, Z    +0.000, E1   +49.402, E3 +44274.364}
SPL {X  -162.871, Y  +348.286, Z    +0.000, E1   +32.462, E3 +44273.392}
SPL {X  -165.127, Y  +365.342, Z    +0.000, E1   +17.250, E3 +44273.230}
SPL {X  -165.640, Y  +376.693, Z    +0.000, E1    +4.721, E3 +44272.803}
SPL {X  -165.650, Y  +380.500, Z    +0.000, E1    -0.000, E3 +44271.954}
SPL {X  -165.650, Y  +383.262, Z    +0.000, E1    -6.645, E3 +44271.483}
SPL {X  -165.650, Y  +388.390, Z    +0.000, E1   -21.508, E3 +44271.271}
SPL {X  -165.650, Y  +393.439, Z    +0.000, E1   -35.398, E3 +44270.839}
SPL {X  -165.650, Y  +400.610, Z    +0.000, E1   -50.510, E3 +44270.576}
SPL {X  -165.650, Y  +414.376, Z    +0.000, E1   -68.098, E3 +44268.610}
SPL {X  -165.650, Y  +468.582, Z    +0.000, E1   -78.237, E3 +44277.380}
SPL {X  -158.306, Y  +724.277, Z    +0.000, E1   -77.461, E3 +44367.821}
ENDSPLINE

SPLINE
SPL {X  -160.145, Y  +717.851, Z    +0.000, E1   -75.386, E3 +44388.335}
ENDSPLINE

SPLINE
SPL {X  -157.156, Y  +727.862, Z    +0.000, E1   -75.175, E3 +44395.807}
SPL {X  -152.814, Y  +739.436, Z    +0.000, E1   -74.813, E3 +44405.660}
SPL {X  -147.104, Y  +751.659, Z    +0.000, E1   -74.255, E3 +44417.105}
SPL {X  -141.453, Y  +761.704, Z    +0.000, E1   -73.638, E3 +44427.318}
SPL {X  -135.914, Y  +770.196, Z    +0.000, E1   -72.974, E3 +44436.379}
SPL {X  -131.459, Y  +776.289, Z    +0.000, E1   -72.475, E3 +44442.455}
SPL {X  -127.605, Y  +781.126, Z    +0.000, E1   -71.922, E3 +44447.899}
SPL {X  -124.773, Y  +784.457, Z    +0.000, E1   -71.383, E3 +44451.947}
SPL {X  -119.086, Y  +790.645, Z    +0.000, E1   -72.931, E3 +44448.801}
SPL {X   -51.449, Y  +832.958, Z    +0.000, E1   -57.230, E3 +44606.321}
ENDSPLINE

SPLINE
SPL {X  -123.821, Y  +785.537, Z    +0.000, E1   -64.536, E3 +44808.066}
SPL {X  -153.467, Y  +737.853, Z    +0.000, E1   -51.757, E3 +44810.381}
SPL {X  -162.176, Y  +709.248, Z    +0.000, E1   -35.773, E3 +44809.406}
SPL {X  -164.888, Y  +691.368, Z    +0.000, E1   -20.174, E3 +44807.844}
SPL {X  -165.597, Y  +679.703, Z    +0.000, E1    -7.645, E3 +44808.019}
SPL {X  -165.650, Y  +673.520, Z    +0.000, E1    -0.048, E3 +44806.971}
SPL {X  -165.650, Y  +671.692, Z    +0.000, E1    +4.450, E3 +44806.537}
SPL {X  -165.650, Y  +667.743, Z    +0.000, E1   +15.617, E3 +44806.455}
SPL {X  -165.650, Y  +661.459, Z    +0.000, E1   +33.218, E3 +44806.035}
SPL {X  -165.650, Y  +653.296, Z    +0.000, E1   +51.333, E3 +44805.591}
SPL {X  -165.650, Y  +642.000, Z    +0.000, E1   +65.561, E3 +44804.803}
SPL {X  -165.650, Y  +619.979, Z    +0.000, E1   +79.465, E3 +44800.810}
SPL {X  -165.650, Y  +584.722, Z    +0.000, E1   +79.551, E3 +44810.100}
SPL {X  -165.650, Y  +560.326, Z    +0.000, E1   +78.360, E3 +44819.823}
SPL {X  -158.840, Y  +331.491, Z    +0.000, E1   +77.462, E3 +44902.398}
ENDSPLINE

SPLINE
SPL {X  -159.893, Y  +335.208, Z    +0.000, E1   +75.483, E3 +44923.133}
ENDSPLINE

SPLINE
SPL {X  -156.487, Y  +324.170, Z    +0.000, E1   +75.150, E3 +44932.514}
SPL {X  -142.256, Y  +293.629, Z    +0.000, E1   +77.020, E3 +44927.614}
ENDSPLINE

SPLINE
SPL {X  -142.811, Y  +294.566, Z    +0.000, E1   +75.668, E3 +44939.576}
ENDSPLINE

SPLINE
SPL {X  -141.646, Y  +292.615, Z    +0.000, E1   +74.702, E3 +44948.670}
SPL {X  -140.419, Y  +290.622, Z    +0.000, E1   +73.705, E3 +44957.513}
SPL {X  -136.008, Y  +283.940, Z    +0.000, E1   +73.594, E3 +44961.632}
SPL {X  -132.748, Y  +279.415, Z    +0.000, E1   +73.006, E3 +44967.688}
SPL {X  -129.007, Y  +274.590, Z    +0.000, E1   +72.484, E3 +44973.037}
SPL {X  -124.646, Y  +269.397, Z    +0.000, E1   +72.041, E3 +44977.785}
SPL {X  -111.023, Y  +255.562, Z    +0.000, E1   +75.772, E3 +44969.567}
SPL {X   -52.752, Y  +221.474, Z    +0.000, E1   +59.157, E3 +45098.818}
SPL {X   -49.901, Y  +220.545, Z    +0.000, E1   +56.696, E3 +45185.211}
ENDSPLINE

SPLINE
SPL {X  -127.117, Y  +272.287, Z    +0.000, E1   +62.713, E3 +45331.503}
SPL {X  -152.442, Y  +313.682, Z    +0.000, E1   +51.943, E3 +45335.735}
SPL {X  -159.925, Y  +335.326, Z    +0.000, E1   +41.361, E3 +45335.677}
SPL {X  -163.450, Y  +351.595, Z    +0.000, E1   +29.785, E3 +45334.789}
SPL {X  -165.127, Y  +365.342, Z    +0.000, E1   +17.250, E3 +45334.769}
SPL {X  -165.640, Y  +376.693, Z    +0.000, E1    +4.721, E3 +45334.342}
SPL {X  -165.650, Y  +380.500, Z    +0.000, E1    -0.000, E3 +45333.493}
SPL {X  -165.650, Y  +383.262, Z    +0.000, E1    -6.645, E3 +45333.022}
SPL {X  -165.650, Y  +388.390, Z    +0.000, E1   -21.508, E3 +45332.809}
SPL {X  -165.650, Y  +393.439, Z    +0.000, E1   -35.398, E3 +45332.377}
SPL {X  -165.650, Y  +400.610, Z    +0.000, E1   -50.510, E3 +45332.115}
SPL {X  -165.650, Y  +414.376, Z    +0.000, E1   -68.098, E3 +45330.148}
SPL {X  -165.650, Y  +468.582, Z    +0.000, E1   -78.237, E3 +45338.918}
SPL {X  -158.306, Y  +724.277, Z    +0.000, E1   -77.461, E3 +45429.360}
ENDSPLINE

SPLINE
SPL {X  -160.145, Y  +717.851, Z    +0.000, E1   -75.386, E3 +45449.873}
ENDSPLINE

SPLINE
SPL {X  -157.156, Y  +727.862, Z    +0.000, E1   -75.175, E3 +45457.345}
SPL {X  -152.814, Y  +739.436, Z    +0.000, E1   -74.813, E3 +45467.199}
SPL {X  -147.104, Y  +751.659, Z    +0.000, E1   -74.255, E3 +45478.643}
SPL {X  -141.453, Y  +761.704, Z    +0.000, E1   -73.638, E3 +45488.856}
SPL {X  -135.914, Y  +770.196, Z    +0.000, E1   -72.974, E3 +45497.918}
SPL {X  -131.459, Y  +776.289, Z    +0.000, E1   -72.475, E3 +45503.994}
SPL {X  -127.605, Y  +781.126, Z    +0.000, E1   -71.922, E3 +45509.438}
SPL {X  -124.773, Y  +784.457, Z    +0.000, E1   -71.383, E3 +45513.485}
SPL {X  -119.086, Y  +790.645, Z    +0.000, E1   -72.931, E3 +45510.339}
SPL {X   -51.449, Y  +832.958, Z    +0.000, E1   -57.230, E3 +45667.859}
ENDSPLINE

SPLINE
SPL {X  -123.821, Y  +785.537, Z    +0.000, E1   -64.536, E3 +45869.604}
SPL {X  -153.467, Y  +737.853, Z    +0.000, E1   -51.757, E3 +45871.919}
SPL {X  -162.176, Y  +709.248, Z    +0.000, E1   -35.773, E3 +45870.945}
SPL {X  -164.888, Y  +691.368, Z    +0.000, E1   -20.174, E3 +45869.382}
SPL {X  -165.597, Y  +679.703, Z    +0.000, E1    -7.645, E3 +45869.557}
SPL {X  -165.650, Y  +673.520, Z    +0.000, E1    -0.048, E3 +45868.509}
SPL {X  -165.650, Y  +671.692, Z    +0.000, E1    +4.450, E3 +45868.076}
SPL {X  -165.650, Y  +667.743, Z    +0.000, E1   +15.617, E3 +45867.994}
SPL {X  -165.650, Y  +661.459, Z    +0.000, E1   +33.218, E3 +45867.574}
SPL {X  -165.650, Y  +653.296, Z    +0.000, E1   +51.333, E3 +45867.129}
SPL {X  -165.650, Y  +642.000, Z    +0.000, E1   +65.561, E3 +45866.341}
SPL {X  -165.650, Y  +619.979, Z    +0.000, E1   +79.465, E3 +45862.348}
SPL {X  -165.650, Y  +584.722, Z    +0.000, E1   +79.551, E3 +45871.639}
SPL {X  -165.650, Y  +560.326, Z    +0.000, E1   +78.360, E3 +45881.361}
SPL {X  -160.258, Y  +336.579, Z    +0.000, E1   +78.314, E3 +45952.883}
SPL {X  -159.618, Y  +334.207, Z    +0.000, E1   +75.622, E3 +45983.697}
SPL {X  -157.855, Y  +328.284, Z    +0.000, E1   +75.167, E3 +45991.662}
SPL {X  -155.139, Y  +320.432, Z    +0.000, E1   +75.106, E3 +45996.339}
SPL {X  -142.256, Y  +293.629, Z    +0.000, E1   +77.020, E3 +45989.152}
ENDSPLINE

SPLINE
SPL {X  -142.811, Y  +294.566, Z    +0.000, E1   +75.668, E3 +46001.115}
ENDSPLINE

SPLINE
SPL {X  -141.646, Y  +292.615, Z    +0.000, E1   +74.702, E3 +46010.208}
SPL {X  -140.419, Y  +290.622, Z    +0.000, E1   +73.705, E3 +46019.052}
SPL {X  -136.008, Y  +283.940, Z    +0.000, E1   +73.594, E3 +46023.171}
SPL {X  -131.988, Y  +278.404, Z    +0.000, E1   +72.860, E3 +46030.725}
SPL {X  -126.848, Y  +271.966, Z    +0.000, E1   +72.322, E3 +46036.770}
SPL {X  -123.729, Y  +268.359, Z    +0.000, E1   +71.932, E3 +46040.239}
SPL {X  -111.023, Y  +255.562, Z    +0.000, E1   +75.772, E3 +46031.105}
SPL {X   -49.289, Y  +220.353, Z    +0.000, E1   +56.690, E3 +46223.820}
ENDSPLINE

SPLINE
SPL {X  -127.117, Y  +272.287, Z    +0.000, E1   +62.713, E3 +46393.042}
SPL {X  -152.442, Y  +313.682, Z    +0.000, E1   +51.943, E3 +46397.274}
SPL {X  -159.925, Y  +335.326, Z    +0.000, E1   +41.361, E3 +46397.216}
SPL {X  -163.450, Y  +351.595, Z    +0.000, E1   +29.785, E3 +46396.327}
SPL {X  -165.127, Y  +365.342, Z    +0.000, E1   +17.250, E3 +46396.307}
SPL {X  -165.640, Y  +376.693, Z    +0.000, E1    +4.721, E3 +46395.880}
SPL {X  -165.650, Y  +380.500, Z    +0.000, E1    -0.000, E3 +46395.031}
SPL {X  -165.650, Y  +382.123, Z    +0.000, E1    -3.912, E3 +46394.658}
SPL {X  -165.650, Y  +387.069, Z    +0.000, E1   -17.420, E3 +46394.370}
SPL {X  -165.650, Y  +393.439, Z    +0.000, E1   -35.398, E3 +46393.915}
SPL {X  -165.650, Y  +402.896, Z    +0.000, E1   -54.480, E3 +46393.157}
SPL {X  -165.650, Y  +416.934, Z    +0.000, E1   -69.887, E3 +46391.623}
SPL {X  -165.650, Y  +459.729, Z    +0.000, E1   -78.035, E3 +46398.141}
SPL {X  -165.650, Y  +475.450, Z    +0.000, E1   -78.345, E3 +46402.255}
SPL {X  -158.306, Y  +724.277, Z    +0.000, E1   -77.461, E3 +46490.898}
ENDSPLINE

SPLINE
SPL {X  -160.145, Y  +717.851, Z    +0.000, E1   -75.386, E3 +46511.412}
ENDSPLINE

SPLINE
SPL {X  -157.156, Y  +727.862, Z    +0.000, E1   -75.175, E3 +46518.884}
SPL {X  -154.068, Y  +736.353, Z    +0.000, E1   -74.906, E3 +46526.058}
SPL {X  -149.738, Y  +746.340, Z    +0.000, E1   -74.451, E3 +46535.746}
SPL {X  -145.204, Y  +755.223, Z    +0.000, E1   -74.188, E3 +46542.472}
SPL {X  -141.453, Y  +761.704, Z    +0.000, E1   -73.638, E3 +46550.395}
SPL {X  -135.914, Y  +770.196, Z    +0.000, E1   -72.974, E3 +46559.456}
SPL {X  -131.459, Y  +776.289, Z    +0.000, E1   -72.475, E3 +46565.532}
SPL {X  -128.771, Y  +779.702, Z    +0.000, E1   -71.875, E3 +46570.479}
SPL {X  -124.506, Y  +784.762, Z    +0.000, E1   -71.815, E3 +46573.367}
SPL {X  -112.958, Y  +796.663, Z    +0.000, E1   -74.119, E3 +46570.071}
SPL {X   -51.449, Y  +832.958, Z    +0.000, E1   -57.230, E3 +46729.398}
ENDSPLINE

SPLINE
SPL {X  -123.821, Y  +785.537, Z    +0.000, E1   -64.536, E3 +46931.143}
SPL {X  -153.467, Y  +737.853, Z    +0.000, E1   -51.757, E3 +46933.458}
SPL {X  -162.176, Y  +709.248, Z    +0.000, E1   -35.773, E3 +46932.483}
SPL {X  -164.888, Y  +691.368, Z    +0.000, E1   -20.174, E3 +46930.921}
SPL {X  -165.597, Y  +679.703, Z    +0.000, E1    -7.645, E3 +46931.096}
SPL {X  -165.650, Y  +673.520, Z    +0.000, E1    -0.048, E3 +46930.048}
SPL {X  -165.650, Y  +671.692, Z    +0.000, E1    +4.450, E3 +46929.614}
SPL {X  -165.650, Y  +667.743, Z    +0.000, E1   +15.617, E3 +46929.532}
SPL {X  -165.650, Y  +661.459, Z    +0.000, E1   +33.218, E3 +46929.112}
SPL {X  -165.650, Y  +653.296, Z    +0.000, E1   +51.333, E3 +46928.668}
SPL {X  -165.650, Y  +642.000, Z    +0.000, E1   +65.561, E3 +46927.880}
SPL {X  -165.650, Y  +619.979, Z    +0.000, E1   +79.465, E3 +46923.886}
SPL {X  -165.650, Y  +569.632, Z    +0.000, E1   +78.783, E3 +46939.165}
SPL {X  -158.840, Y  +331.491, Z    +0.000, E1   +77.462, E3 +47025.475}
ENDSPLINE

SPLINE
SPL {X  -159.893, Y  +335.208, Z    +0.000, E1   +75.483, E3 +47046.210}
ENDSPLINE

SPLINE
SPL {X  -156.487, Y  +324.170, Z    +0.000, E1   +75.150, E3 +47055.591}
SPL {X  -142.256, Y  +293.629, Z    +0.000, E1   +77.020, E3 +47050.691}
ENDSPLINE

SPLINE
SPL {X  -142.811, Y  +294.566, Z    +0.000, E1   +75.668, E3 +47062.653}
ENDSPLINE

SPLINE
SPL {X  -141.646, Y  +292.615, Z    +0.000, E1   +74.702, E3 +47071.747}
SPL {X  -140.419, Y  +290.622, Z    +0.000, E1   +73.705, E3 +47080.590}
SPL {X  -135.839, Y  +283.697, Z    +0.000, E1   +73.388, E3 +47086.328}
SPL {X  -131.336, Y  +277.551, Z    +0.000, E1   +72.879, E3 +47092.581}
SPL {X  -126.848, Y  +271.966, Z    +0.000, E1   +72.322, E3 +47098.309}
SPL {X  -123.729, Y  +268.359, Z    +0.000, E1   +71.932, E3 +47101.778}
SPL {X  -111.023, Y  +255.562, Z    +0.000, E1   +75.772, E3 +47092.644}
SPL {X   -52.752, Y  +221.474, Z    +0.000, E1   +59.157, E3 +47221.895}
SPL {X   -49.901, Y  +220.545, Z    +0.000, E1   +56.696, E3 +47308.288}
ENDSPLINE

SPLINE
SPL {X  -127.117, Y  +272.287, Z    +0.000, E1   +62.713, E3 +47454.580}
SPL {X  -152.442, Y  +313.682, Z    +0.000, E1   +51.943, E3 +47458.812}
SPL {X  -162.319, Y  +345.447, Z    +0.000, E1   +34.671, E3 +47458.238}
SPL {X  -165.127, Y  +365.342, Z    +0.000, E1   +17.250, E3 +47457.846}
SPL {X  -165.640, Y  +376.693, Z    +0.000, E1    +4.721, E3 +47457.419}
SPL {X  -165.650, Y  +380.500, Z    +0.000, E1    -0.000, E3 +47456.569}
SPL {X  -165.650, Y  +382.123, Z    +0.000, E1    -3.912, E3 +47456.197}
SPL {X  -165.650, Y  +387.069, Z    +0.000, E1   -17.420, E3 +47455.908}
SPL {X  -165.650, Y  +393.439, Z    +0.000, E1   -35.398, E3 +47455.454}
SPL {X  -165.650, Y  +400.610, Z    +0.000, E1   -50.510, E3 +47455.192}
SPL {X  -165.650, Y  +414.376, Z    +0.000, E1   -68.098, E3 +47453.225}
SPL {X  -165.650, Y  +468.582, Z    +0.000, E1   -78.237, E3 +47461.995}
SPL {X  -160.244, Y  +717.475, Z    +0.000, E1   -78.917, E3 +47534.553}
SPL {X  -159.651, Y  +719.676, Z    +0.000, E1   -75.661, E3 +47570.940}
SPL {X  -157.156, Y  +727.862, Z    +0.000, E1   -75.175, E3 +47580.422}
SPL {X  -154.068, Y  +736.353, Z    +0.000, E1   -74.906, E3 +47587.597}
SPL {X  -149.738, Y  +746.340, Z    +0.000, E1   -74.451, E3 +47597.284}
SPL {X  -144.163, Y  +757.090, Z    +0.000, E1   -74.033, E3 +47606.377}
SPL {X  -139.284, Y  +765.165, Z    +0.000, E1   -73.322, E3 +47616.072}
SPL {X  -134.662, Y  +771.969, Z    +0.000, E1   -72.884, E3 +47622.403}
SPL {X  -131.459, Y  +776.289, Z    +0.000, E1   -72.475, E3 +47627.070}
SPL {X  -127.605, Y  +781.126, Z    +0.000, E1   -71.922, E3 +47632.515}
SPL {X  -124.773, Y  +784.457, Z    +0.000, E1   -71.383, E3 +47636.562}
SPL {X  -119.086, Y  +790.645, Z    +0.000, E1   -72.931, E3 +47633.416}
SPL {X   -51.449, Y  +832.958, Z    +0.000, E1   -57.230, E3 +47790.936}
ENDSPLINE

SPLINE
SPL {X  -123.821, Y  +785.537, Z    +0.000, E1   -64.536, E3 +47992.681}
SPL {X  -153.467, Y  +737.853, Z    +0.000, E1   -51.757, E3 +47994.996}
SPL {X  -161.000, Y  +714.475, Z    +0.000, E1   -39.424, E3 +47994.469}
SPL {X  -164.534, Y  +694.695, Z    +0.000, E1   -23.511, E3 +47992.759}
SPL {X  -165.597, Y  +679.703, Z    +0.000, E1    -7.645, E3 +47992.634}
SPL {X  -165.650, Y  +673.520, Z    +0.000, E1    -0.048, E3 +47991.586}
SPL {X  -165.650, Y  +671.692, Z    +0.000, E1    +4.450, E3 +47991.153}
SPL {X  -165.650, Y  +667.743, Z    +0.000, E1   +15.617, E3 +47991.070}
SPL {X  -165.650, Y  +661.459, Z    +0.000, E1   +33.218, E3 +47990.651}
SPL {X  -165.650, Y  +653.296, Z    +0.000, E1   +51.333, E3 +47990.206}
SPL {X  -165.650, Y  +642.000, Z    +0.000, E1   +65.561, E3 +47989.418}
SPL {X  -165.650, Y  +619.979, Z    +0.000, E1   +79.465, E3 +47985.425}
SPL {X  -165.650, Y  +569.632, Z    +0.000, E1   +78.783, E3 +48000.704}
SPL {X  -158.840, Y  +331.491, Z    +0.000, E1   +77.462, E3 +48087.014}
ENDSPLINE

SPLINE
SPL {X  -159.893, Y  +335.208, Z    +0.000, E1   +75.483, E3 +48107.748}
ENDSPLINE

SPLINE
SPL {X  -156.487, Y  +324.170, Z    +0.000, E1   +75.150, E3 +48117.130}
SPL {X  -142.256, Y  +293.629, Z    +0.000, E1   +77.020, E3 +48112.229}
ENDSPLINE

SPLINE
SPL {X  -142.811, Y  +294.566, Z    +0.000, E1   +75.668, E3 +48124.192}
ENDSPLINE

SPLINE
SPL {X  -141.646, Y  +292.615, Z    +0.000, E1   +74.702, E3 +48133.285}
SPL {X  -140.419, Y  +290.622, Z    +0.000, E1   +73.705, E3 +48142.129}
SPL {X  -136.008, Y  +283.940, Z    +0.000, E1   +73.594, E3 +48146.248}
SPL {X  -132.748, Y  +279.415, Z    +0.000, E1   +73.006, E3 +48152.303}
SPL {X  -129.007, Y  +274.590, Z    +0.000, E1   +72.484, E3 +48157.652}
SPL {X  -125.914, Y  +270.864, Z    +0.000, E1   +72.144, E3 +48161.144}
SPL {X  -123.729, Y  +268.359, Z    +0.000, E1   +71.932, E3 +48163.316}
SPL {X  -111.023, Y  +255.562, Z    +0.000, E1   +75.772, E3 +48154.182}
SPL {X   -49.289, Y  +220.353, Z    +0.000, E1   +56.690, E3 +48346.897}
ENDSPLINE

SPLINE
SPL {X  -127.117, Y  +272.287, Z    +0.000, E1   +62.713, E3 +48516.119}
SPL {X  -154.956, Y  +319.945, Z    +0.000, E1   +49.402, E3 +48520.518}
SPL {X  -162.871, Y  +348.286, Z    +0.000, E1   +32.462, E3 +48519.546}
SPL {X  -165.127, Y  +365.342, Z    +0.000, E1   +17.250, E3 +48519.384}
SPL {X  -165.640, Y  +376.693, Z    +0.000, E1    +4.721, E3 +48518.957}
SPL {X  -165.650, Y  +380.500, Z    +0.000, E1    -0.000, E3 +48518.108}
SPL {X  -165.650, Y  +382.123, Z    +0.000, E1    -3.912, E3 +48517.735}
SPL {X  -165.650, Y  +387.069, Z    +0.000, E1   -17.420, E3 +48517.447}
SPL {X  -165.650, Y  +393.439, Z    +0.000, E1   -35.398, E3 +48516.992}
SPL {X  -165.650, Y  +402.896, Z    +0.000, E1   -54.480, E3 +48516.234}
SPL {X  -165.650, Y  +416.934, Z    +0.000, E1   -69.887, E3 +48514.700}
SPL {X  -165.650, Y  +459.729, Z    +0.000, E1   -78.035, E3 +48521.218}
SPL {X  -165.650, Y  +475.450, Z    +0.000, E1   -78.345, E3 +48525.332}
SPL {X  -160.244, Y  +717.475, Z    +0.000, E1   -78.917, E3 +48596.092}
SPL {X  -159.651, Y  +719.676, Z    +0.000, E1   -75.661, E3 +48632.478}
SPL {X  -157.156, Y  +727.862, Z    +0.000, E1   -75.175, E3 +48641.961}
SPL {X  -154.068, Y  +736.353, Z    +0.000, E1   -74.906, E3 +48649.135}
SPL {X  -149.738, Y  +746.340, Z    +0.000, E1   -74.451, E3 +48658.823}
SPL {X  -144.163, Y  +757.090, Z    +0.000, E1   -74.033, E3 +48667.915}
SPL {X  -139.284, Y  +765.165, Z    +0.000, E1   -73.322, E3 +48677.610}
SPL {X  -134.662, Y  +771.969, Z    +0.000, E1   -72.884, E3 +48683.942}
SPL {X  -131.459, Y  +776.289, Z    +0.000, E1   -72.475, E3 +48688.609}
SPL {X  -128.771, Y  +779.702, Z    +0.000, E1   -71.875, E3 +48693.556}
SPL {X  -125.267, Y  +783.889, Z    +0.000, E1   -71.674, E3 +48696.668}
SPL {X  -119.086, Y  +790.645, Z    +0.000, E1   -72.931, E3 +48694.955}
SPL {X   -51.449, Y  +832.958, Z    +0.000, E1   -57.230, E3 +48852.475}
ENDSPLINE

SPLINE
SPL {X  -123.821, Y  +785.537, Z    +0.000, E1   -64.536, E3 +49054.220}
SPL {X  -153.467, Y  +737.853, Z    +0.000, E1   -51.757, E3 +49056.534}
SPL {X  -162.176, Y  +709.248, Z    +0.000, E1   -35.773, E3 +49055.560}
SPL {X  -164.888, Y  +691.368, Z    +0.000, E1   -20.174, E3 +49053.998}
SPL {X  -165.597, Y  +679.703, Z    +0.000, E1    -7.645, E3 +49054.173}
SPL {X  -165.650, Y  +673.520, Z    +0.000, E1    -0.048, E3 +49053.124}
SPL {X  -165.650, Y  +671.692, Z    +0.000, E1    +4.450, E3 +49052.691}
SPL {X  -165.650, Y  +667.743, Z    +0.000, E1   +15.617, E3 +49052.609}
SPL {X  -165.650, Y  +661.459, Z    +0.000, E1   +33.218, E3 +49052.189}
SPL {X  -165.650, Y  +653.296, Z    +0.000, E1   +51.333, E3 +49051.745}
SPL {X  -165.650, Y  +642.000, Z    +0.000, E1   +65.561, E3 +49050.957}
SPL {X  -165.650, Y  +619.979, Z    +0.000, E1   +79.465, E3 +49046.963}
SPL {X  -165.650, Y  +584.722, Z    +0.000, E1   +79.551, E3 +49056.254}
SPL {X  -165.650, Y  +560.326, Z    +0.000, E1   +78.360, E3 +49065.977}
SPL {X  -158.840, Y  +331.491, Z    +0.000, E1   +77.462, E3 +49148.552}
ENDSPLINE

SPLINE
SPL {X  -159.893, Y  +335.208, Z    +0.000, E1   +75.483, E3 +49169.287}
ENDSPLINE

SPLINE
SPL {X  -156.487, Y  +324.170, Z    +0.000, E1   +75.150, E3 +49178.668}
SPL {X  -142.256, Y  +293.629, Z    +0.000, E1   +77.020, E3 +49173.768}
ENDSPLINE

SPLINE
SPL {X  -142.811, Y  +294.566, Z    +0.000, E1   +75.668, E3 +49185.730}
ENDSPLINE

SPLINE
SPL {X  -141.646, Y  +292.615, Z    +0.000, E1   +74.702, E3 +49194.824}
SPL {X  -140.419, Y  +290.622, Z    +0.000, E1   +73.705, E3 +49203.667}
SPL {X  -136.008, Y  +283.940, Z    +0.000, E1   +73.594, E3 +49207.786}
SPL {X  -132.748, Y  +279.415, Z    +0.000, E1   +73.006, E3 +49213.842}
SPL {X  -129.007, Y  +274.590, Z    +0.000, E1   +72.484, E3 +49219.191}
SPL {X  -125.914, Y  +270.864, Z    +0.000, E1   +72.144, E3 +49222.682}
SPL {X  -123.729, Y  +268.359, Z    +0.000, E1   +71.932, E3 +49224.855}
SPL {X  -111.023, Y  +255.562, Z    +0.000, E1   +75.772, E3 +49215.720}
SPL {X   -49.289, Y  +220.353, Z    +0.000, E1   +56.690, E3 +49408.435}
ENDSPLINE

SPLINE
SPL {X  -127.117, Y  +272.287, Z    +0.000, E1   +62.713, E3 +49577.657}
SPL {X  -152.442, Y  +313.682, Z    +0.000, E1   +51.943, E3 +49581.889}
SPL {X  -159.925, Y  +335.326, Z    +0.000, E1   +41.361, E3 +49581.831}
SPL {X  -163.450, Y  +351.595, Z    +0.000, E1   +29.785, E3 +49580.942}
SPL {X  -165.127, Y  +365.342, Z    +0.000, E1   +17.250, E3 +49580.923}
SPL {X  -165.640, Y  +376.693, Z    +0.000, E1    +4.721, E3 +49580.496}
SPL {X  -165.650, Y  +380.500, Z    +0.000, E1    -0.000, E3 +49579.646}
SPL {X  -165.650, Y  +382.123, Z    +0.000, E1    -3.912, E3 +49579.274}
SPL {X  -165.650, Y  +387.069, Z    +0.000, E1   -17.420, E3 +49578.985}
SPL {X  -165.650, Y  +393.439, Z    +0.000, E1   -35.398, E3 +49578.531}
SPL {X  -165.650, Y  +400.610, Z    +0.000, E1   -50.510, E3 +49578.268}
SPL {X  -165.650, Y  +414.376, Z    +0.000, E1   -68.098, E3 +49576.302}
SPL {X  -165.650, Y  +468.582, Z    +0.000, E1   -78.237, E3 +49585.072}
SPL {X  -160.244, Y  +717.475, Z    +0.000, E1   -78.917, E3 +49657.630}
SPL {X  -159.651, Y  +719.676, Z    +0.000, E1   -75.661, E3 +49694.017}
SPL {X  -157.156, Y  +727.862, Z    +0.000, E1   -75.175, E3 +49703.499}
SPL {X  -152.814, Y  +739.436, Z    +0.000, E1   -74.813, E3 +49713.353}
SPL {X  -148.754, Y  +748.385, Z    +0.000, E1   -74.281, E3 +49722.795}
SPL {X  -144.163, Y  +757.090, Z    +0.000, E1   -74.033, E3 +49729.454}
SPL {X  -140.473, Y  +763.291, Z    +0.000, E1   -73.478, E3 +49736.895}
SPL {X  -135.914, Y  +770.196, Z    +0.000, E1   -72.974, E3 +49744.072}
SPL {X  -131.459, Y  +776.289, Z    +0.000, E1   -72.475, E3 +49750.147}
SPL {X  -128.771, Y  +779.702, Z    +0.000, E1   -71.875, E3 +49755.094}
SPL {X  -125.267, Y  +783.889, Z    +0.000, E1   -71.674, E3 +49758.206}
SPL {X  -119.086, Y  +790.645, Z    +0.000, E1   -72.931, E3 +49756.493}
SPL {X   -51.449, Y  +832.958, Z    +0.000, E1   -57.230, E3 +49914.013}
ENDSPLINE

SPLINE
SPL {X  -123.821, Y  +785.537, Z    +0.000, E1   -64.536, E3 +50115.758}
SPL {X  -153.467, Y  +737.853, Z    +0.000, E1   -51.757, E3 +50118.073}
SPL {X  -161.000, Y  +714.475, Z    +0.000, E1   -39.424, E3 +50117.546}
SPL {X  -164.534, Y  +694.695, Z    +0.000, E1   -23.511, E3 +50115.835}
SPL {X  -165.597, Y  +679.703, Z    +0.000, E1    -7.645, E3 +50115.711}
SPL {X  -165.650, Y  +673.520, Z    +0.000, E1    -0.048, E3 +50114.663}
SPL {X  -165.650, Y  +671.692, Z    +0.000, E1    +4.450, E3 +50114.230}
SPL {X  -165.650, Y  +667.743, Z    +0.000, E1   +15.617, E3 +50114.147}
SPL {X  -165.650, Y  +662.891, Z    +0.000, E1   +29.740, E3 +50113.665}
SPL {X  -165.650, Y  +655.319, Z    +0.000, E1   +47.265, E3 +50113.514}
SPL {X  -165.650, Y  +642.000, Z    +0.000, E1   +65.561, E3 +50112.495}
SPL {X  -165.650, Y  +619.979, Z    +0.000, E1   +79.465, E3 +50108.502}
SPL {X  -165.650, Y  +569.632, Z    +0.000, E1   +78.783, E3 +50123.781}
SPL {X  -158.840, Y  +331.491, Z    +0.000, E1   +77.462, E3 +50210.091}
ENDSPLINE

SPLINE
SPL {X  -159.893, Y  +335.208, Z    +0.000, E1   +75.483, E3 +50230.825}
ENDSPLINE

SPLINE
SPL {X  -156.487, Y  +324.170, Z    +0.000, E1   +75.150, E3 +50240.207}
SPL {X  -142.256, Y  +293.629, Z    +0.000, E1   +77.020, E3 +50235.306}
ENDSPLINE

SPLINE
SPL {X  -142.811, Y  +294.566, Z    +0.000, E1   +75.668, E3 +50247.269}
ENDSPLINE

SPLINE
SPL {X  -141.646, Y  +292.615, Z    +0.000, E1   +74.702, E3 +50256.362}
SPL {X  -140.419, Y  +290.622, Z    +0.000, E1   +73.705, E3 +50265.205}
SPL {X  -135.839, Y  +283.697, Z    +0.000, E1   +73.388, E3 +50270.944}
SPL {X  -131.903, Y  +278.292, Z    +0.000, E1   +73.096, E3 +50275.433}
SPL {X  -129.007, Y  +274.590, Z    +0.000, E1   +72.484, E3 +50280.729}
SPL {X  -124.646, Y  +269.397, Z    +0.000, E1   +72.041, E3 +50285.477}
SPL {X  -111.023, Y  +255.562, Z    +0.000, E1   +75.772, E3 +50277.259}
SPL {X   -49.289, Y  +220.353, Z    +0.000, E1   +56.690, E3 +50469.974}
ENDSPLINE

SPLINE
SPL {X  -127.117, Y  +272.287, Z    +0.000, E1   +62.713, E3 +50639.196}
SPL {X  -154.956, Y  +319.945, Z    +0.000, E1   +49.402, E3 +50643.595}
SPL {X  -162.871, Y  +348.286, Z    +0.000, E1   +32.462, E3 +50642.623}
SPL {X  -165.127, Y  +365.342, Z    +0.000, E1   +17.250, E3 +50642.461}
SPL {X  -165.640, Y  +376.693, Z    +0.000, E1    +4.721, E3 +50642.034}
SPL {X  -165.650, Y  +380.500, Z    +0.000, E1    -0.000, E3 +50641.185}
SPL {X  -165.650, Y  +383.262, Z    +0.000, E1    -6.645, E3 +50640.714}
SPL {X  -165.650, Y  +388.390, Z    +0.000, E1   -21.508, E3 +50640.502}
SPL {X  -165.650, Y  +393.439, Z    +0.000, E1   -35.398, E3 +50640.069}
SPL {X  -165.650, Y  +400.610, Z    +0.000, E1   -50.510, E3 +50639.807}
SPL {X  -165.650, Y  +414.376, Z    +0.000, E1   -68.098, E3 +50637.841}
SPL {X  -165.650, Y  +468.582, Z    +0.000, E1   -78.237, E3 +50646.611}
SPL {X  -158.306, Y  +724.277, Z    +0.000, E1   -77.461, E3 +50737.052}
ENDSPLINE

SPLINE
SPL {X  -160.145, Y  +717.851, Z    +0.000, E1   -75.386, E3 +50757.565}
ENDSPLINE

SPLINE
SPL {X  -157.156, Y  +727.862, Z    +0.000, E1   -75.175, E3 +50765.038}
SPL {X  -154.068, Y  +736.353, Z    +0.000, E1   -74.906, E3 +50772.212}
SPL {X  -149.738, Y  +746.340, Z    +0.000, E1   -74.451, E3 +50781.900}
SPL {X  -144.163, Y  +757.090, Z    +0.000, E1   -74.033, E3 +50790.992}
SPL {X  -140.473, Y  +763.291, Z    +0.000, E1   -73.478, E3 +50798.434}
SPL {X  -135.914, Y  +770.196, Z    +0.000, E1   -72.974, E3 +50805.610}
SPL {X  -131.459, Y  +776.289, Z    +0.000, E1   -72.475, E3 +50811.686}
SPL {X  -128.771, Y  +779.702, Z    +0.000, E1   -71.875, E3 +50816.632}
SPL {X  -124.506, Y  +784.762, Z    +0.000, E1   -71.815, E3 +50819.521}
SPL {X  -112.958, Y  +796.663, Z    +0.000, E1   -74.119, E3 +50816.224}
SPL {X   -51.449, Y  +832.958, Z    +0.000, E1   -57.230, E3 +50975.551}
ENDSPLINE

SPLINE
SPL {X  -123.821, Y  +785.537, Z    +0.000, E1   -64.536, E3 +51177.297}
SPL {X  -153.467, Y  +737.853, Z    +0.000, E1   -51.757, E3 +51179.611}
SPL {X  -162.176, Y  +709.248, Z    +0.000, E1   -35.773, E3 +51178.637}
SPL {X  -164.888, Y  +691.368, Z    +0.000, E1   -20.174, E3 +51177.075}
SPL {X  -165.597, Y  +679.703, Z    +0.000, E1    -7.645, E3 +51177.250}
SPL {X  -165.650, Y  +673.520, Z    +0.000, E1    -0.048, E3 +51176.201}
SPL {X  -165.650, Y  +671.692, Z    +0.000, E1    +4.450, E3 +51175.768}
SPL {X  -165.650, Y  +667.743, Z    +0.000, E1   +15.617, E3 +51175.686}
SPL {X  -165.650, Y  +661.459, Z    +0.000, E1   +33.218, E3 +51175.266}
SPL {X  -165.650, Y  +650.834, Z    +0.000, E1   +55.143, E3 +51174.654}
SPL {X  -165.650, Y  +639.785, Z    +0.000, E1   +67.512, E3 +51173.871}
SPL {X  -165.650, Y  +619.979, Z    +0.000, E1   +79.465, E3 +51170.040}
SPL {X  -165.650, Y  +569.632, Z    +0.000, E1   +78.783, E3 +51185.319}
SPL {X  -158.840, Y  +331.491, Z    +0.000, E1   +77.462, E3 +51271.629}
ENDSPLINE

SPLINE
SPL {X  -159.893, Y  +335.208, Z    +0.000, E1   +75.483, E3 +51292.364}
ENDSPLINE

SPLINE
SPL {X  -156.487, Y  +324.170, Z    +0.000, E1   +75.150, E3 +51301.745}
SPL {X  -142.256, Y  +293.629, Z    +0.000, E1   +77.020, E3 +51296.845}
ENDSPLINE

SPLINE
SPL {X  -142.811, Y  +294.566, Z    +0.000, E1   +75.668, E3 +51308.807}
ENDSPLINE

SPLINE
SPL {X  -141.646, Y  +292.615, Z    +0.000, E1   +74.702, E3 +51317.901}
SPL {X  -140.419, Y  +290.622, Z    +0.000, E1   +73.705, E3 +51326.744}
SPL {X  -136.008, Y  +283.940, Z    +0.000, E1   +73.594, E3 +51330.863}
SPL {X  -132.748, Y  +279.415, Z    +0.000, E1   +73.006, E3 +51336.919}
SPL {X  -129.007, Y  +274.590, Z    +0.000, E1   +72.484, E3 +51342.268}
SPL {X  -125.914, Y  +270.864, Z    +0.000, E1   +72.144, E3 +51345.759}
SPL {X  -123.729, Y  +268.359, Z    +0.000, E1   +71.932, E3 +51347.932}
SPL {X  -111.023, Y  +255.562, Z    +0.000, E1   +75.772, E3 +51338.797}
SPL {X   -49.289, Y  +220.353, Z    +0.000, E1   +56.690, E3 +51531.512}
ENDSPLINE

SPLINE
SPL {X  -127.117, Y  +272.287, Z    +0.000, E1   +62.713, E3 +51700.734}
SPL {X  -154.956, Y  +319.945, Z    +0.000, E1   +49.402, E3 +51705.133}
SPL {X  -162.871, Y  +348.286, Z    +0.000, E1   +32.462, E3 +51704.161}
SPL {X  -165.127, Y  +365.342, Z    +0.000, E1   +17.250, E3 +51704.000}
SPL {X  -165.640, Y  +376.693, Z    +0.000, E1    +4.721, E3 +51703.572}
SPL {X  -165.650, Y  +380.500, Z    +0.000, E1    -0.000, E3 +51702.723}
SPL {X  -165.650, Y  +383.262, Z    +0.000, E1    -6.645, E3 +51702.253}
SPL {X  -165.650, Y  +388.390, Z    +0.000, E1   -21.508, E3 +51702.040}
SPL {X  -165.650, Y  +393.439, Z    +0.000, E1   -35.398, E3 +51701.608}
SPL {X  -165.650, Y  +400.610, Z    +0.000, E1   -50.510, E3 +51701.345}
SPL {X  -165.650, Y  +414.376, Z    +0.000, E1   -68.098, E3 +51699.379}
SPL {X  -165.650, Y  +468.582, Z    +0.000, E1   -78.237, E3 +51708.149}
SPL {X  -158.306, Y  +724.277, Z    +0.000, E1   -77.461, E3 +51798.591}
ENDSPLINE

SPLINE
SPL {X  -160.145, Y  +717.851, Z    +0.000, E1   -75.386, E3 +51819.104}
ENDSPLINE

SPLINE
SPL {X  -157.156, Y  +727.862, Z    +0.000, E1   -75.175, E3 +51826.576}
SPL {X  -152.814, Y  +739.436, Z    +0.000, E1   -74.813, E3 +51836.430}
SPL {X  -148.754, Y  +748.385, Z    +0.000, E1   -74.281, E3 +51845.872}
SPL {X  -144.163, Y  +757.090, Z    +0.000, E1   -74.033, E3 +51852.531}
SPL {X  -140.473, Y  +763.291, Z    +0.000, E1   -73.478, E3 +51859.972}
SPL {X  -135.914, Y  +770.196, Z    +0.000, E1   -72.974, E3 +51867.148}
SPL {X  -131.459, Y  +776.289, Z    +0.000, E1   -72.475, E3 +51873.224}
SPL {X  -128.771, Y  +779.702, Z    +0.000, E1   -71.875, E3 +51878.171}
SPL {X  -125.267, Y  +783.889, Z    +0.000, E1   -71.674, E3 +51881.283}
SPL {X  -119.086, Y  +790.645, Z    +0.000, E1   -72.931, E3 +51879.570}
SPL {X   -51.449, Y  +832.958, Z    +0.000, E1   -57.230, E3 +52037.090}
ENDSPLINE

SPLINE
SPL {X  -113.713, Y  +795.955, Z    +0.000, E1   -65.735, E3 +52236.008}
SPL {X  -131.116, Y  +776.736, Z    +0.000, E1   -63.149, E3 +52240.538}
SPL {X  -153.467, Y  +737.853, Z    +0.000, E1   -51.757, E3 +52241.150}
SPL {X  -161.000, Y  +714.475, Z    +0.000, E1   -39.424, E3 +52240.622}
SPL {X  -164.534, Y  +694.695, Z    +0.000, E1   -23.511, E3 +52238.912}
SPL {X  -165.597, Y  +679.703, Z    +0.000, E1    -7.645, E3 +52238.788}
SPL {X  -165.650, Y  +673.520, Z    +0.000, E1    -0.048, E3 +52237.740}
SPL {X  -165.650, Y  +671.692, Z    +0.000, E1    +4.450, E3 +52237.306}
SPL {X  -165.650, Y  +667.743, Z    +0.000, E1   +15.617, E3 +52237.224}
SPL {X  -165.650, Y  +661.459, Z    +0.000, E1   +33.218, E3 +52236.805}
SPL {X  -165.650, Y  +653.296, Z    +0.000, E1   +51.333, E3 +52236.360}
SPL {X  -165.650, Y  +642.000, Z    +0.000, E1   +65.561, E3 +52235.572}
SPL {X  -165.650, Y  +619.979, Z    +0.000, E1   +79.465, E3 +52231.579}
SPL {X  -165.650, Y  +584.722, Z    +0.000, E1   +79.551, E3 +52240.870}
SPL {X  -165.650, Y  +560.326, Z    +0.000, E1   +78.360, E3 +52250.592}
SPL {X  -160.258, Y  +336.579, Z    +0.000, E1   +78.314, E3 +52322.114}
SPL {X  -159.618, Y  +334.207, Z    +0.000, E1   +75.622, E3 +52352.928}
SPL {X  -157.855, Y  +328.284, Z    +0.000, E1   +75.167, E3 +52360.893}
SPL {X  -155.139, Y  +320.432, Z    +0.000, E1   +75.106, E3 +52365.570}
SPL {X  -142.256, Y  +293.629, Z    +0.000, E1   +77.020, E3 +52358.383}
ENDSPLINE

SPLINE
SPL {X  -142.811, Y  +294.566, Z    +0.000, E1   +75.668, E3 +52370.346}
ENDSPLINE

SPLINE
SPL {X  -141.646, Y  +292.615, Z    +0.000, E1   +74.702, E3 +52379.439}
SPL {X  -140.419, Y  +290.622, Z    +0.000, E1   +73.705, E3 +52388.282}
SPL {X  -136.008, Y  +283.940, Z    +0.000, E1   +73.594, E3 +52392.401}
SPL {X  -131.988, Y  +278.404, Z    +0.000, E1   +72.860, E3 +52399.956}
SPL {X  -126.848, Y  +271.966, Z    +0.000, E1   +72.322, E3 +52406.001}
SPL {X  -123.729, Y  +268.359, Z    +0.000, E1   +71.932, E3 +52409.470}
SPL {X  -111.023, Y  +255.562, Z    +0.000, E1   +75.772, E3 +52400.336}
SPL {X   -49.289, Y  +220.353, Z    +0.000, E1   +56.690, E3 +52593.051}
ENDSPLINE

SPLINE
SPL {X  -127.117, Y  +272.287, Z    +0.000, E1   +62.713, E3 +52762.273}
SPL {X  -152.442, Y  +313.682, Z    +0.000, E1   +51.943, E3 +52766.505}
SPL {X  -162.319, Y  +345.447, Z    +0.000, E1   +34.671, E3 +52765.930}
SPL {X  -165.127, Y  +365.342, Z    +0.000, E1   +17.250, E3 +52765.538}
SPL {X  -165.640, Y  +376.693, Z    +0.000, E1    +4.721, E3 +52765.111}
SPL {X  -165.650, Y  +380.500, Z    +0.000, E1    -0.000, E3 +52764.262}
SPL {X  -165.650, Y  +383.262, Z    +0.000, E1    -6.645, E3 +52763.791}
SPL {X  -165.650, Y  +388.390, Z    +0.000, E1   -21.508, E3 +52763.579}
SPL {X  -165.650, Y  +393.439, Z    +0.000, E1   -35.398, E3 +52763.146}
SPL {X  -165.650, Y  +400.610, Z    +0.000, E1   -50.510, E3 +52762.884}
SPL {X  -165.650, Y  +414.376, Z    +0.000, E1   -68.098, E3 +52760.917}
SPL {X  -165.650, Y  +468.582, Z    +0.000, E1   -78.237, E3 +52769.688}
SPL {X  -158.306, Y  +724.277, Z    +0.000, E1   -77.461, E3 +52860.129}
ENDSPLINE

SPLINE
SPL {X  -160.145, Y  +717.851, Z    +0.000, E1   -75.386, E3 +52880.642}
ENDSPLINE

SPLINE
SPL {X  -157.156, Y  +727.862, Z    +0.000, E1   -75.175, E3 +52888.114}
SPL {X  -152.814, Y  +739.436, Z    +0.000, E1   -74.813, E3 +52897.968}
SPL {X  -147.104, Y  +751.659, Z    +0.000, E1   -74.255, E3 +52909.413}
SPL {X  -141.453, Y  +761.704, Z    +0.000, E1   -73.638, E3 +52919.625}
SPL {X  -135.914, Y  +770.196, Z    +0.000, E1   -72.974, E3 +52928.687}
SPL {X  -131.459, Y  +776.289, Z    +0.000, E1   -72.475, E3 +52934.763}
SPL {X  -127.605, Y  +781.126, Z    +0.000, E1   -71.922, E3 +52940.207}
SPL {X  -124.773, Y  +784.457, Z    +0.000, E1   -71.383, E3 +52944.254}
SPL {X  -119.086, Y  +790.645, Z    +0.000, E1   -72.931, E3 +52941.109}
SPL {X   -51.449, Y  +832.958, Z    +0.000, E1   -57.230, E3 +53098.628}
ENDSPLINE

